// TIA Portal project "acesys_wincc_faceplates" (V16)

(* hardware
DEVICE "PC-System_1"  SIMATIC PC station
   slot 0: "SIMATIC PC station"  Rail  SIMATIC PC-Station  V1.0
      slot 125: "Stationmanager"  Station_Manager  V6.0.4
   slot 1: "HMI_RT_1"  WinCC RT Professional  6AV2 105-0xxxx-xxxx  16.0.0.0
*)

(* ===== HMI "HMI_RT_1" =====
system functions are stored by id; their names below are inferred from use
connection "994": S71200_TCP_IP, SCADA_S7_1500_OMS
connection "993": S71200_TCP_IP, SCADA_S7_1500_OMS
connection "995": S71200_TCP_IP, SCADA_S7_1500_OMS
connection "996": S71200_TCP_IP, SCADA_S7_1500_OMS
connection "997": S71200_TCP_IP, SCADA_S7_1500_OMS

HMI tags "Default tag table"
   "HMI_Tag_1" : Int, internal
   "vis_tab_int" : Int, internal
   "status_ord" : Int, internal

HMI tags "020PU043U01"
   "020PU043U01.BlockInfo" : Array [0..4] of Int AT %DB4312.DBX74.0, 500 ms
   "020PU043U01.FP_CMD" : Int AT %DB4312.DBW84, 500 ms
   "020PU043U01.FP_DIM.Auto" : Bool AT %DB4312.DBX92.0, 500 ms
   "020PU043U01.FP_DIM" : Array [0..15] of Bool AT %DB4312.DBX92.0, 500 ms
   "020PU043U01.FP_SHOW" : Array [0..15] of Bool AT %DB4312.DBX94.0, 500 ms
   "020PU043U01.FP_SHOW_1" : Int AT %DB4312.DBW96, 500 ms
   "020PU043U01.FP_SHOW.PB_Auto" : Bool AT %DB4312.DBX94.0, 500 ms
   "020PU043U01.FP_SHOW.PB_Local" : Bool AT %DB4312.DBX94.1, 500 ms
   "020PU043U01.FP_SHOW.PB_Manual" : Bool AT %DB4312.DBX94.2, 500 ms
   "020PU043U01.FP_SHOW.PB_Start1" : Bool AT %DB4312.DBX94.3, 500 ms
   "020PU043U01.FP_SHOW.PB_Start2" : Bool AT %DB4312.DBX94.4, 500 ms
   "020PU043U01.FP_SHOW.PB_Stop" : Bool AT %DB4312.DBX94.5, 500 ms
   "020PU043U01.FP_SHOW.PB_Test" : Bool AT %DB4312.DBX94.6, 500 ms
   "020PU043U01.FP_SHOW.PB_QStop" : Bool AT %DB4312.DBX94.7, 500 ms
   "020PU043U01.FP_SHOW.AI1" : Bool AT %DB4312.DBX95.0, 500 ms
   "020PU043U01.FP_SHOW.AI2" : Bool AT %DB4312.DBX95.1, 500 ms
   "020PU043U01.FP_SHOW.AI3" : Bool AT %DB4312.DBX95.2, 500 ms
   "020PU043U01.FP_SHOW.SP" : Bool AT %DB4312.DBX95.3, 500 ms
   "020PU043U01.FP_SHOW.MCC" : Bool AT %DB4312.DBX95.4, 500 ms
   "020PU043U01.FP_SHOW.RDY" : Bool AT %DB4312.DBX95.5, 500 ms
   "020PU043U01.FP_SHOW.OVL" : Bool AT %DB4312.DBX95.6, 500 ms
   "020PU043U01.FP_SHOW.LSTP" : Bool AT %DB4312.DBX95.7, 500 ms
   "020PU043U01.FP_SHOW.REM" : Bool AT %DB4312.DBX96.0, 500 ms
   "020PU043U01.FP_SHOW.SSW" : Bool AT %DB4312.DBX96.1, 500 ms
   "020PU043U01.FP_SHOW.ES" : Bool AT %DB4312.DBX96.2, 500 ms
   "020PU043U01.FP_SHOW.TFA" : Bool AT %DB4312.DBX96.3, 500 ms
   "020PU043U01.FP_SHOW.DRDY" : Bool AT %DB4312.DBX96.4, 500 ms
   "020PU043U01.FP_SHOW.STALL" : Bool AT %DB4312.DBX96.5, 500 ms
   "020PU043U01.FP_SHOW.EARTH" : Bool AT %DB4312.DBX96.6, 500 ms
   "020PU043U01.FP_SHOW.UBAL" : Bool AT %DB4312.DBX96.7, 500 ms
   "020PU043U01.FP_SHOW.GFA" : Bool AT %DB4312.DBX97.0, 500 ms
   "020PU043U01.FP_SHOW.GWA" : Bool AT %DB4312.DBX97.1, 500 ms
   "020PU043U01.FP_SHOW.BUSF" : Bool AT %DB4312.DBX97.2, 500 ms
   "020PU043U01.FP_SHOW.DOPR" : Bool AT %DB4312.DBX97.3, 500 ms
   "020PU043U01.FP_SHOW.DTEST" : Bool AT %DB4312.DBX97.4, 500 ms
   "020PU043U01.FP_SHOW.ACK" : Bool AT %DB4312.DBX97.5, 500 ms
   "020PU043U01.FP_SHOW.LSTR1" : Bool AT %DB4312.DBX97.6, 500 ms
   "020PU043U01.FP_SHOW.LSTR2" : Bool AT %DB4312.DBX97.7, 500 ms
   "020PU043U01.FP_SHOW.RET2" : Bool AT %DB4312.DBX98.0, 500 ms
   "020PU043U01.FP_SHOW.RUN2" : Bool AT %DB4312.DBX98.1, 500 ms
   "020PU043U01.FP_SHOW.CON2" : Bool AT %DB4312.DBX98.2, 500 ms
   "020PU043U01.FP_SHOW.RD2" : Bool AT %DB4312.DBX98.3, 500 ms
   "020PU043U01.FP_SHOW.SFS" : Bool AT %DB4312.DBX98.4, 500 ms
   "020PU043U01.FP_SHOW.SLS" : Bool AT %DB4312.DBX98.5, 500 ms
   "020PU043U01.FP_SHOW.MD" : Bool AT %DB4312.DBX98.6, 500 ms
   "020PU043U01.FP_SHOW.DelayRun2" : Bool AT %DB4312.DBX98.7, 500 ms
   "020PU043U01.FP_SHOW.ChangeDir" : Bool AT %DB4312.DBX99.0, 500 ms
   "020PU043U01.FP_SHOW.PB_Reset" : Bool AT %DB4312.DBX99.1, 500 ms
   "020PU043U01.FP_SHOW.ASTR" : Bool AT %DB4312.DBX99.2, 500 ms
   "020PU043U01.FP_PARM.StartWarn_Pre" : Int AT %DB4312.DBW100, 500 ms
   "020PU043U01.FP_PARM.StartWarn_Acc" : Int AT %DB4312.DBW102, 500 ms
   "020PU043U01.FP_PARM.RunDelay1_Pre" : Int AT %DB4312.DBW104, 500 ms
   "020PU043U01.FP_PARM.RunDelay1_Acc" : Int AT %DB4312.DBW106, 500 ms
   "020PU043U01.FP_PARM.RunDelay2_Pre" : Int AT %DB4312.DBW108, 500 ms
   "020PU043U01.FP_PARM.RunDelay2_Acc" : Int AT %DB4312.DBW110, 500 ms
   "020PU043U01.FP_PARM.DelayStart_Pre" : Int AT %DB4312.DBW112, 500 ms
   "020PU043U01.FP_PARM.DelayStart_Acc" : Int AT %DB4312.DBW114, 500 ms
   "020PU043U01.FP_PARM.DelayStop_Pre" : Int AT %DB4312.DBW116, 500 ms
   "020PU043U01.FP_PARM.DelayStop_Acc" : Int AT %DB4312.DBW118, 500 ms
   "020PU043U01.FP_PARM.ReturnMon_Pre" : Int AT %DB4312.DBW120, 500 ms
   "020PU043U01.FP_PARM.ReturnMon_Acc" : Int AT %DB4312.DBW122, 500 ms
   "020PU043U01.FP_PARM.SpeedMonOnDelay_Pre" : Int AT %DB4312.DBW124, 500 ms
   "020PU043U01.FP_PARM.SpeedMonOnDelay_Acc" : Int AT %DB4312.DBW126, 500 ms
   "020PU043U01.FP_PARM.SpeedMonOffDelay_Pre" : Int AT %DB4312.DBW128, 500 ms
   "020PU043U01.FP_PARM.SpeedMonOffDelay_Acc" : Int AT %DB4312.DBW130, 500 ms
   "020PU043U01.FP_PARM.SpeedMonTrigDelay_Pre" : Int AT %DB4312.DBW132, 500 ms
   "020PU043U01.FP_PARM.SpeedMonTrigDelay_Acc" : Int AT %DB4312.DBW134, 500 ms
   "020PU043U01.FP_PARM.ChangeDir_Pre" : Int AT %DB4312.DBW136, 500 ms
   "020PU043U01.FP_PARM.ChangeDir_Acc" : Int AT %DB4312.DBW138, 500 ms
   "020PU043U01.FP_PARM.LeaveFS_Pre" : Int AT %DB4312.DBW140, 500 ms
   "020PU043U01.FP_PARM.LeaveFS_Acc" : Int AT %DB4312.DBW142, 500 ms
   "020PU043U01.FP_PARM.ReachLS_Pre" : Int AT %DB4312.DBW144, 500 ms
   "020PU043U01.FP_PARM.ReachLS_Acc" : Int AT %DB4312.DBW146, 500 ms
   "020PU043U01.FP_PARM.ReachFS_Pre" : Int AT %DB4312.DBW148, 500 ms
   "020PU043U01.FP_PARM.ReachFS_Acc" : Int AT %DB4312.DBW150, 500 ms
   "020PU043U01.FP_PARM.MD_Freq_SP" : Int AT %DB4312.DBW152, 500 ms
   "020PU043U01.FP_PARM.MD_Freq_PV" : Int AT %DB4312.DBW154, 500 ms
   "020PU043U01.FP_PARM.StopReason" : Bool AT %DB4312.DBX156.0, 500 ms
   "020PU043U01.FP_PARM.AI1_Max" : Real AT %DB4312.DBD158, 500 ms
   "020PU043U01.FP_PARM.AI1_Min" : Real AT %DB4312.DBD162, 500 ms
   "020PU043U01.FP_PARM.AI2_Max" : Real AT %DB4312.DBD166, 500 ms
   "020PU043U01.FP_PARM.AI2_Min" : Real AT %DB4312.DBD170, 500 ms
   "020PU043U01.FP_PARM.AI3_Max" : Real AT %DB4312.DBD174, 500 ms
   "020PU043U01.FP_PARM.AI3_Min" : Real AT %DB4312.DBD178, 500 ms
   "020PU043U01.FP_PARM.AO1a_Max" : Real AT %DB4312.DBD182, 500 ms
   "020PU043U01.FP_PARM.AO1a_Min" : Real AT %DB4312.DBD186, 500 ms
   "020PU043U01.FP_PARM.AO2a_Max" : Real AT %DB4312.DBD190, 500 ms
   "020PU043U01.FP_PARM.AO2a_Min" : Real AT %DB4312.DBD194, 500 ms
   "020PU043U01.FP_PARM.AO3a_Max" : Real AT %DB4312.DBD198, 500 ms
   "020PU043U01.FP_PARM.AO3a_Min" : Real AT %DB4312.DBD202, 500 ms
   "020PU043U01.FP_PARM.AO1b_Max" : Real AT %DB4312.DBD206, 500 ms
   "020PU043U01.FP_PARM.AO1b_Min" : Real AT %DB4312.DBD210, 500 ms
   "020PU043U01.FP_PARM.AO2b_Max" : Real AT %DB4312.DBD214, 500 ms
   "020PU043U01.FP_PARM.AO2b_Min" : Real AT %DB4312.DBD218, 500 ms
   "020PU043U01.FP_PARM.AO3b_Max" : Real AT %DB4312.DBD222, 500 ms
   "020PU043U01.FP_PARM.AO3b_Min" : Real AT %DB4312.DBD226, 500 ms
   "020PU043U01.FP_PARM.INTL" : Bool AT %DB4312.DBX230.0, 500 ms
   "020PU043U01.FP_PARM.INTL_SEQ_STR1" : Bool AT %DB4312.DBX230.1, 500 ms
   "020PU043U01.FP_PARM.INTL_SEQ_STR2" : Bool AT %DB4312.DBX230.2, 500 ms
   "020PU043U01.FP_PARM.INTL_SEQ_STP" : Bool AT %DB4312.DBX230.3, 500 ms
   "020PU043U01.StatusWork" : Int AT %DB4312.DBW494, 500 ms
   "020PU043U01.ModePointer" : Int AT %DB4312.DBW496, 500 ms
   "020PU043U01.AO1b" : Real AT %DB4312.DBD38, 500 ms
   "020PU043U01.AO2b" : Real AT %DB4312.DBD46, 500 ms
   "020PU043U01.AO3b" : Real AT %DB4312.DBD54, 500 ms
   "020PU043U01.SPSET" : Real AT %DB4312.DBD18, 500 ms
   "020PU043U01.AO3a" : Real AT %DB4312.DBD50, 500 ms
   "020PU043U01.AO2a" : Real AT %DB4312.DBD42, 500 ms
   "020PU043U01.AO1a" : Real AT %DB4312.DBD34, 500 ms
   "020PU043U01.FP_DIM.FP_DIM" : Bool AT %DB4312.DBX92.0, 500 ms
   "020PU043U01.FP_DIM.Local" : Bool AT %DB4312.DBX92.1, 500 ms
   "020PU043U01.FP_DIM.Manual" : Bool AT %DB4312.DBX92.2, 500 ms
   "020PU043U01.FP_DIM.Start1" : Bool AT %DB4312.DBX92.3, 500 ms
   "020PU043U01.FP_DIM.Start2" : Bool AT %DB4312.DBX92.4, 500 ms
   "020PU043U01.FP_DIM.Stop" : Bool AT %DB4312.DBX92.5, 500 ms
   "020PU043U01.FP_DIM.TEst" : Bool AT %DB4312.DBX92.6, 500 ms
   "020PU043U01.FP_DIM.QStop" : Bool AT %DB4312.DBX92.7, 500 ms
   "020PU043U01.FP_DIM.Reset" : Bool AT %DB4312.DBX93.0, 500 ms
   "020PU043U01.FP_EN.Mode_Auto" : Bool AT %DB4312.DBX90.0, 500 ms
   "020PU043U01.FP_EN.Mode_Man" : Bool AT %DB4312.DBX90.1, 500 ms
   "020PU043U01.FP_EN.Mode_Loc" : Bool AT %DB4312.DBX90.2, 500 ms
   "020PU043U01.FP_EN.Mode_Test" : Bool AT %DB4312.DBX90.3, 500 ms
   "020PU043U01.FP_EN.Mode_SS_Field" : Bool AT %DB4312.DBX90.4, 500 ms
   "020PU043U01.FP_EN.Mode_SS_FP" : Bool AT %DB4312.DBX90.5, 500 ms
   "020PU043U01.FP_EN.PB_QStop" : Bool AT %DB4312.DBX90.6, 500 ms
   "020PU043U01.FP_CMD.QuickStop" : Bool AT %DB4312.DBX84.0, 500 ms
   "020PU043U01.FP_CMD.AckAlarm" : Bool AT %DB4312.DBX84.7, 500 ms
   "020PU043U01.FP_CMD.Auto" : Bool AT %DB4312.DBX85.0, 500 ms
   "020PU043U01.FP_CMD.Manual" : Bool AT %DB4312.DBX85.1, 500 ms
   "020PU043U01.FP_CMD.Local" : Bool AT %DB4312.DBX85.2, 500 ms
   "020PU043U01.FP_CMD.Start1" : Bool AT %DB4312.DBX85.3, 500 ms
   "020PU043U01.FP_CMD.Start2" : Bool AT %DB4312.DBX85.4, 500 ms
   "020PU043U01.FP_CMD.Stop" : Bool AT %DB4312.DBX85.5, 500 ms
   "020PU043U01.FP_CMD.Reset" : Bool AT %DB4312.DBX85.6, 500 ms
   "020PU043U01.FP_CMD.Test" : Bool AT %DB4312.DBX85.7, 500 ms
   "020PU043U01.DI.SEL" : Bool AT %DB4312.DBX2.0, 500 ms
   "020PU043U01.DI.ASTR" : Bool AT %DB4312.DBX2.1, 500 ms
   "020PU043U01.DI.DIR" : Bool AT %DB4312.DBX2.2, 500 ms
   "020PU043U01.DI.MCC" : Bool AT %DB4312.DBX2.3, 500 ms
   "020PU043U01.DI.RDY" : Bool AT %DB4312.DBX2.4, 500 ms
   "020PU043U01.DI.OVL" : Bool AT %DB4312.DBX2.5, 500 ms
   "020PU043U01.DI.RET1" : Bool AT %DB4312.DBX2.6, 500 ms
   "020PU043U01.DI.RET2" : Bool AT %DB4312.DBX2.7, 500 ms
   "020PU043U01.DI.LSTR1" : Bool AT %DB4312.DBX3.0, 500 ms
   "020PU043U01.DI.LSTR2" : Bool AT %DB4312.DBX3.1, 500 ms
   "020PU043U01.DI.LSTP" : Bool AT %DB4312.DBX3.2, 500 ms
   "020PU043U01.DI.REM" : Bool AT %DB4312.DBX3.3, 500 ms
   "020PU043U01.DI.SSW" : Bool AT %DB4312.DBX3.4, 500 ms
   "020PU043U01.DI.TFA" : Bool AT %DB4312.DBX3.5, 500 ms
   "020PU043U01.DI.DRDY" : Bool AT %DB4312.DBX3.6, 500 ms
   "020PU043U01.DI.MD" : Bool AT %DB4312.DBX3.7, 500 ms
   "020PU043U01.DI.STALL" : Bool AT %DB4312.DBX4.0, 500 ms
   "020PU043U01.DI.EARTH" : Bool AT %DB4312.DBX4.1, 500 ms
   "020PU043U01.DI.UBAL" : Bool AT %DB4312.DBX4.2, 500 ms
   "020PU043U01.DI.GFA" : Bool AT %DB4312.DBX4.3, 500 ms
   "020PU043U01.DI.GWA" : Bool AT %DB4312.DBX4.4, 500 ms
   "020PU043U01.DI.BUSF" : Bool AT %DB4312.DBX4.5, 500 ms
   "020PU043U01.DI.DOPR" : Bool AT %DB4312.DBX4.6, 500 ms
   "020PU043U01.DI.DTEST" : Bool AT %DB4312.DBX4.7, 500 ms
   "020PU043U01.DI.SFS" : Bool AT %DB4312.DBX5.0, 500 ms
   "020PU043U01.DI.SLS" : Bool AT %DB4312.DBX5.1, 500 ms
   "020PU043U01.DI.ES" : Bool AT %DB4312.DBX5.2, 500 ms
   "020PU043U01.DI.ACK" : Bool AT %DB4312.DBX5.3, 500 ms
   "020PU043U01.DQ.CON1" : Bool AT %DB4312.DBX30.0, 500 ms
   "020PU043U01.DQ.CON2" : Bool AT %DB4312.DBX30.1, 500 ms
   "020PU043U01.DQ.LAMP1" : Bool AT %DB4312.DBX30.2, 500 ms
   "020PU043U01.DQ.LAMP2" : Bool AT %DB4312.DBX30.3, 500 ms
   "020PU043U01.DQ.SACK" : Bool AT %DB4312.DBX30.4, 500 ms
   "020PU043U01.DQ.RD1" : Bool AT %DB4312.DBX30.5, 500 ms
   "020PU043U01.DQ.RD2" : Bool AT %DB4312.DBX30.6, 500 ms
   "020PU043U01.DQ.RUN1" : Bool AT %DB4312.DBX30.7, 500 ms
   "020PU043U01.DQ.RUN2" : Bool AT %DB4312.DBX31.0, 500 ms
   "020PU043U01.DQ.OK" : Bool AT %DB4312.DBX31.1, 500 ms
   "020PU043U01.DQ.LOC" : Bool AT %DB4312.DBX31.2, 500 ms
   "020PU043U01.DQ.MAN" : Bool AT %DB4312.DBX31.3, 500 ms
   "020PU043U01.DQ.AUT" : Bool AT %DB4312.DBX31.4, 500 ms
   "020PU043U01.DQ.SS" : Bool AT %DB4312.DBX31.5, 500 ms
   "020PU043U01.DQ.RES" : Bool AT %DB4312.DBX31.6, 500 ms
   "020PU043U01.DQ.TESTP" : Bool AT %DB4312.DBX31.7, 500 ms
   "020PU043U01.DQ.ASTW" : Bool AT %DB4312.DBX32.0, 500 ms
   "020PU043U01.AI1" : Real AT %DB4312.DBD6, 500 ms
   "020PU043U01.AI2" : Real AT %DB4312.DBD10, 500 ms
   "020PU043U01.AI3" : Real AT %DB4312.DBD14, 500 ms
   "020PU043U01.FP_SEL.MD" : Bool AT %DB4312.DBX86.0, 500 ms
   "020PU043U01.FP_SEL.MD_Puls" : Bool AT %DB4312.DBX86.1, 500 ms
   "020PU043U01.FP_SEL.MD_OnOff" : Bool AT %DB4312.DBX86.2, 500 ms
   "020PU043U01.FP_SEL.MD_Maintain" : Bool AT %DB4312.DBX86.3, 500 ms
   "020PU043U01.FP_SEL.STW_AutoStart" : Bool AT %DB4312.DBX86.4, 500 ms
   "020PU043U01.FP_SEL.STW_Local" : Bool AT %DB4312.DBX86.5, 500 ms
   "020PU043U01.FP_SEL.STW_Manual" : Bool AT %DB4312.DBX86.6, 500 ms
   "020PU043U01.FP_SEL.STW_Single" : Bool AT %DB4312.DBX86.7, 500 ms
   "020PU043U01.FP_SEL.Type_Unimotor" : Bool AT %DB4312.DBX87.0, 500 ms
   "020PU043U01.FP_SEL.Type_Bimotor" : Bool AT %DB4312.DBX87.1, 500 ms
   "020PU043U01.FP_SEL.Type_Indication" : Bool AT %DB4312.DBX87.2, 500 ms
   "020PU043U01.FP_SEL.MotorStarter" : Bool AT %DB4312.DBX87.3, 500 ms
   "020PU043U01.FP_SEL.ParentSupress" : Bool AT %DB4312.DBX87.4, 500 ms
   "020PU043U01.FP_SEL.ParentCollection" : Bool AT %DB4312.DBX87.5, 500 ms
   "020PU043U01.FP_SEL.INCH_Man" : Bool AT %DB4312.DBX87.6, 500 ms
   "020PU043U01.FP_SEL.INCH_Loc" : Bool AT %DB4312.DBX87.7, 500 ms
   "020PU043U01.FP_SEL.OutOfSevice" : Bool AT %DB4312.DBX88.0, 500 ms
   "020PU043U01.FP_SEL.WarningDrive" : Bool AT %DB4312.DBX88.1, 500 ms
   "020PU043U01.FP_SHOW.B1" : Byte AT %DB4313.DBB95, 500 ms
   "020PU043U01.FP_SHOW.B2" : Byte AT %DB4313.DBB96, 500 ms
   "020PU043U01.FP_SHOW.B3" : Byte AT %DB4313.DBB97, 500 ms
   "020PU043U01.FP_SHOW.B4" : Byte AT %DB4313.DBB98, 500 ms
   "020PU043U01.FP_SHOW.B5" : Byte AT %DB4313.DBB99, 500 ms
   "020PU043U01.MSW" : DWord AT %DB4312.DBD62, 500 ms
   "020PU043U01.ParentInfo" : String[10], internal
   "020PU043U01.DefaultText" : String[32], internal   // Заголовок POPUP окна. При експорте из ECS через скрипт заполняется автоматически, если теги копируются в ручную то требуется в ручную задатать свойство Start Value

HMI tags "020PU044U01"
   "020PU044U01.BlockInfo" : Array [0..4] of Int AT %DB4313.DBX74.0, 500 ms
   "020PU044U01.FP_CMD" : Int AT %DB4313.DBW84, 500 ms
   "020PU044U01.MSW" : DWord AT %DB4313.DBD62, 500 ms
   "020PU044U01.FP_DIM.Auto" : Bool AT %DB4313.DBX92.0, 500 ms
   "020PU044U01.FP_DIM1" : Array [0..15] of Bool AT %DB4313.DBX92.0, 500 ms
   "020PU044U01.FP_SHOW" : Array [0..15] of Bool AT %DB4313.DBX94.0, 500 ms
   "020PU044U01.FP_SHOW_1" : Int AT %DB4313.DBW96, 500 ms
   "020PU044U01.FP_SHOW.PB_Auto" : Bool AT %DB4313.DBX94.0, 500 ms
   "020PU044U01.FP_SHOW.PB_Local" : Bool AT %DB4313.DBX94.1, 500 ms
   "020PU044U01.FP_SHOW.PB_Manual" : Bool AT %DB4313.DBX94.2, 500 ms
   "020PU044U01.FP_SHOW.PB_Start1" : Bool AT %DB4313.DBX94.3, 500 ms
   "020PU044U01.FP_SHOW.PB_Start2" : Bool AT %DB4313.DBX94.4, 500 ms
   "020PU044U01.FP_SHOW.PB_Stop" : Bool AT %DB4313.DBX94.5, 500 ms
   "020PU044U01.FP_SHOW.PB_Test" : Bool AT %DB4313.DBX94.6, 500 ms
   "020PU044U01.FP_SHOW.PB_QStop" : Bool AT %DB4313.DBX94.7, 500 ms
   "020PU044U01.FP_SHOW.AI1" : Bool AT %DB4313.DBX95.0, 500 ms
   "020PU044U01.FP_SHOW.AI2" : Bool AT %DB4313.DBX95.1, 500 ms
   "020PU044U01.FP_SHOW.AI3" : Bool AT %DB4313.DBX95.2, 500 ms
   "020PU044U01.FP_SHOW.SP" : Bool AT %DB4313.DBX95.3, 500 ms
   "020PU044U01.FP_SHOW.MCC" : Bool AT %DB4313.DBX95.4, 500 ms
   "020PU044U01.FP_SHOW.RDY" : Bool AT %DB4313.DBX95.5, 500 ms
   "020PU044U01.FP_SHOW.OVL" : Bool AT %DB4313.DBX95.6, 500 ms
   "020PU044U01.FP_SHOW.LSTP" : Bool AT %DB4313.DBX95.7, 500 ms
   "020PU044U01.FP_SHOW.REM" : Bool AT %DB4313.DBX96.0, 500 ms
   "020PU044U01.FP_SHOW.SSW" : Bool AT %DB4313.DBX96.1, 500 ms
   "020PU044U01.FP_SHOW.ES" : Bool AT %DB4313.DBX96.2, 500 ms
   "020PU044U01.FP_SHOW.TFA" : Bool AT %DB4313.DBX96.3, 500 ms
   "020PU044U01.FP_SHOW.DRDY" : Bool AT %DB4313.DBX96.4, 500 ms
   "020PU044U01.FP_SHOW.STALL" : Bool AT %DB4313.DBX96.5, 500 ms
   "020PU044U01.FP_SHOW.EARTH" : Bool AT %DB4313.DBX96.6, 500 ms
   "020PU044U01.FP_SHOW.UBAL" : Bool AT %DB4313.DBX96.7, 500 ms
   "020PU044U01.FP_SHOW.GFA" : Bool AT %DB4313.DBX97.0, 500 ms
   "020PU044U01.FP_SHOW.GWA" : Bool AT %DB4313.DBX97.1, 500 ms
   "020PU044U01.FP_SHOW.BUSF" : Bool AT %DB4313.DBX97.2, 500 ms
   "020PU044U01.FP_SHOW.DOPR" : Bool AT %DB4313.DBX97.3, 500 ms
   "020PU044U01.FP_SHOW.DTEST" : Bool AT %DB4313.DBX97.4, 500 ms
   "020PU044U01.FP_SHOW.ACK" : Bool AT %DB4313.DBX97.5, 500 ms
   "020PU044U01.FP_SHOW.LSTR1" : Bool AT %DB4313.DBX97.6, 500 ms
   "020PU044U01.FP_SHOW.LSTR2" : Bool AT %DB4313.DBX97.7, 500 ms
   "020PU044U01.FP_SHOW.RET2" : Bool AT %DB4313.DBX98.0, 500 ms
   "020PU044U01.FP_SHOW.RUN2" : Bool AT %DB4313.DBX98.1, 500 ms
   "020PU044U01.FP_SHOW.CON2" : Bool AT %DB4313.DBX98.2, 500 ms
   "020PU044U01.FP_SHOW.RD2" : Bool AT %DB4313.DBX98.3, 500 ms
   "020PU044U01.FP_SHOW.SFS" : Bool AT %DB4313.DBX98.4, 500 ms
   "020PU044U01.FP_SHOW.SLS" : Bool AT %DB4313.DBX98.5, 500 ms
   "020PU044U01.FP_SHOW.MD" : Bool AT %DB4313.DBX98.6, 500 ms
   "020PU044U01.FP_SHOW.DelayRun2" : Bool AT %DB4313.DBX98.7, 500 ms
   "020PU044U01.FP_SHOW.ChangeDir" : Bool AT %DB4313.DBX99.0, 500 ms
   "020PU044U01.FP_SHOW.PB_Reset" : Bool AT %DB4313.DBX99.1, 500 ms
   "020PU044U01.FP_SHOW.ASTR" : Bool AT %DB4313.DBX99.2, 500 ms
   "020PU044U01.FP_PARM.StartWarn_Pre" : Int AT %DB4313.DBW100, 500 ms
   "020PU044U01.FP_PARM.StartWarn_Acc" : Int AT %DB4313.DBW102, 500 ms
   "020PU044U01.FP_PARM.RunDelay1_Pre" : Int AT %DB4313.DBW104, 500 ms
   "020PU044U01.FP_PARM.RunDelay1_Acc" : Int AT %DB4313.DBW106, 500 ms
   "020PU044U01.FP_PARM.RunDelay2_Pre" : Int AT %DB4313.DBW108, 500 ms
   "020PU044U01.FP_PARM.RunDelay2_Acc" : Int AT %DB4313.DBW110, 500 ms
   "020PU044U01.FP_PARM.DelayStart_Pre" : Int AT %DB4313.DBW112, 500 ms
   "020PU044U01.FP_PARM.DelayStart_Acc" : Int AT %DB4313.DBW114, 500 ms
   "020PU044U01.FP_PARM.DelayStop_Pre" : Int AT %DB4313.DBW116, 500 ms
   "020PU044U01.FP_PARM.DelayStop_Acc" : Int AT %DB4313.DBW118, 500 ms
   "020PU044U01.FP_PARM.ReturnMon_Pre" : Int AT %DB4313.DBW120, 500 ms
   "020PU044U01.FP_PARM.ReturnMon_Acc" : Int AT %DB4313.DBW122, 500 ms
   "020PU044U01.FP_PARM.SpeedMonOnDelay_Pre" : Int AT %DB4313.DBW124, 500 ms
   "020PU044U01.FP_PARM.SpeedMonOnDelay_Acc" : Int AT %DB4313.DBW126, 500 ms
   "020PU044U01.FP_PARM.SpeedMonOffDelay_Pre" : Int AT %DB4313.DBW128, 500 ms
   "020PU044U01.FP_PARM.SpeedMonOffDelay_Acc" : Int AT %DB4313.DBW130, 500 ms
   "020PU044U01.FP_PARM.SpeedMonTrigDelay_Pre" : Int AT %DB4313.DBW132, 500 ms
   "020PU044U01.FP_PARM.SpeedMonTrigDelay_Acc" : Int AT %DB4313.DBW134, 500 ms
   "020PU044U01.FP_PARM.ChangeDir_Pre" : Int AT %DB4313.DBW136, 500 ms
   "020PU044U01.FP_PARM.ChangeDir_Acc" : Int AT %DB4313.DBW138, 500 ms
   "020PU044U01.FP_PARM.LeaveFS_Pre" : Int AT %DB4313.DBW140, 500 ms
   "020PU044U01.FP_PARM.LeaveFS_Acc" : Int AT %DB4313.DBW142, 500 ms
   "020PU044U01.FP_PARM.ReachLS_Pre" : Int AT %DB4313.DBW144, 500 ms
   "020PU044U01.FP_PARM.ReachLS_Acc" : Int AT %DB4313.DBW146, 500 ms
   "020PU044U01.FP_PARM.ReachFS_Pre" : Int AT %DB4313.DBW148, 500 ms
   "020PU044U01.FP_PARM.ReachFS_Acc" : Int AT %DB4313.DBW150, 500 ms
   "020PU044U01.FP_PARM.MD_Freq_SP" : Int AT %DB4313.DBW152, 500 ms
   "020PU044U01.FP_PARM.MD_Freq_PV" : Int AT %DB4313.DBW154, 500 ms
   "020PU044U01.FP_PARM.StopReason" : Int AT %DB4313.DBW156, 500 ms
   "020PU044U01.FP_PARM.AI1_Max" : Real AT %DB4313.DBD158, 500 ms
   "020PU044U01.FP_PARM.AI1_Min" : Real AT %DB4313.DBD162, 500 ms
   "020PU044U01.FP_PARM.AI2_Max" : Real AT %DB4313.DBD166, 500 ms
   "020PU044U01.FP_PARM.AI2_Min" : Real AT %DB4313.DBD170, 500 ms
   "020PU044U01.FP_PARM.AI3_Max" : Real AT %DB4313.DBD174, 500 ms
   "020PU044U01.FP_PARM.AI3_Min" : Real AT %DB4313.DBD178, 500 ms
   "020PU044U01.FP_PARM.AO1a_Max" : Real AT %DB4313.DBD182, 500 ms
   "020PU044U01.FP_PARM.AO1a_Min" : Real AT %DB4313.DBD186, 500 ms
   "020PU044U01.FP_PARM.AO2a_Max" : Real AT %DB4313.DBD190, 500 ms
   "020PU044U01.FP_PARM.AO2a_Min" : Real AT %DB4313.DBD194, 500 ms
   "020PU044U01.FP_PARM.AO3a_Max" : Real AT %DB4313.DBD198, 500 ms
   "020PU044U01.FP_PARM.AO3a_Min" : Real AT %DB4313.DBD202, 500 ms
   "020PU044U01.FP_PARM.AO1b_Max" : Real AT %DB4313.DBD206, 500 ms
   "020PU044U01.FP_PARM.AO1b_Min" : Real AT %DB4313.DBD210, 500 ms
   "020PU044U01.FP_PARM.AO2b_Max" : Real AT %DB4313.DBD214, 500 ms
   "020PU044U01.FP_PARM.AO2b_Min" : Real AT %DB4313.DBD218, 500 ms
   "020PU044U01.FP_PARM.AO3b_Max" : Real AT %DB4313.DBD222, 500 ms
   "020PU044U01.FP_PARM.AO3b_Min" : Real AT %DB4313.DBD226, 500 ms
   "020PU044U01.FP_PARM.INTL" : Bool AT %DB4313.DBX230.0, 500 ms
   "020PU044U01.FP_PARM.INTL_SEQ_STR1" : Bool AT %DB4313.DBX230.1, 500 ms
   "020PU044U01.FP_PARM.INTL_SEQ_STR2" : Bool AT %DB4313.DBX230.2, 500 ms
   "020PU044U01.FP_PARM.INTL_SEQ_STP" : Bool AT %DB4313.DBX230.3, 500 ms
   "020PU044U01.StatusWork" : Int AT %DB4313.DBW494, 500 ms
   "020PU044U01.ModePointer" : Int AT %DB4313.DBW496, 500 ms
   "020PU044U01.AO1b" : Real AT %DB4313.DBD38, 500 ms
   "020PU044U01.AO2b" : Real AT %DB4313.DBD42, 500 ms
   "020PU044U01.AO3b" : Real AT %DB4313.DBD46, 500 ms
   "020PU044U01.SPSET" : Real AT %DB4313.DBD18, 500 ms
   "020PU044U01.AO3a" : Real AT %DB4313.DBD50, 500 ms
   "020PU044U01.AO2a" : Real AT %DB4313.DBD42, 500 ms
   "020PU044U01.AO1a" : Real AT %DB4313.DBD34, 500 ms
   "020PU044U01.FP_DIM.FP_DIM" : Bool AT %DB4313.DBX92.0, 500 ms
   "020PU044U01.FP_DIM.Local" : Bool AT %DB4313.DBX92.1, 500 ms
   "020PU044U01.FP_DIM.Manual" : Bool AT %DB4313.DBX92.2, 500 ms
   "020PU044U01.FP_DIM.Start1" : Bool AT %DB4313.DBX92.3, 500 ms
   "020PU044U01.FP_DIM.Start2" : Bool AT %DB4313.DBX92.4, 500 ms
   "020PU044U01.FP_DIM.Stop" : Bool AT %DB4313.DBX92.5, 500 ms
   "020PU044U01.FP_DIM.TEst" : Bool AT %DB4313.DBX92.6, 500 ms
   "020PU044U01.FP_DIM.QStop" : Bool AT %DB4313.DBX92.7, 500 ms
   "020PU044U01.FP_DIM.Reset" : Bool AT %DB4313.DBX93.0, 500 ms
   "020PU044U01.FP_EN.Mode_Auto" : Bool AT %DB4313.DBX90.0, 500 ms
   "020PU044U01.FP_EN.Mode_Man" : Bool AT %DB4313.DBX90.1, 500 ms
   "020PU044U01.FP_EN.Mode_Loc" : Bool AT %DB4313.DBX90.2, 500 ms
   "020PU044U01.FP_EN.Mode_Test" : Bool AT %DB4313.DBX90.3, 500 ms
   "020PU044U01.FP_EN.Mode_SS_Field" : Bool AT %DB4313.DBX90.4, 500 ms
   "020PU044U01.FP_EN.Mode_SS_FP" : Bool AT %DB4313.DBX90.5, 500 ms
   "020PU044U01.FP_EN.PB_QStop" : Bool AT %DB4313.DBX90.6, 500 ms
   "020PU044U01.FP_EN.Mode_Loc_1" : Bool AT %DB4313.DBX90.3, 500 ms
   "020PU044U01.FP_CMD.QuickStop" : Bool AT %DB4313.DBX84.0, 500 ms
   "020PU044U01.FP_CMD.AckAlarm" : Bool AT %DB4313.DBX84.7, 500 ms
   "020PU044U01.FP_CMD.Auto" : Bool AT %DB4313.DBX85.0, 500 ms
   "020PU044U01.FP_CMD.Manual" : Bool AT %DB4313.DBX85.1, 500 ms
   "020PU044U01.FP_CMD.Local" : Bool AT %DB4313.DBX85.2, 500 ms
   "020PU044U01.FP_CMD.Start1" : Bool AT %DB4313.DBX85.3, 500 ms
   "020PU044U01.FP_CMD.Start2" : Bool AT %DB4313.DBX85.4, 500 ms
   "020PU044U01.FP_CMD.Stop" : Bool AT %DB4313.DBX85.5, 500 ms
   "020PU044U01.FP_CMD.Reset" : Bool AT %DB4313.DBX85.6, 500 ms
   "020PU044U01.FP_CMD.Test" : Bool AT %DB4313.DBX85.7, 500 ms
   "020PU044U01.DI.SEL" : Bool AT %DB4313.DBX2.0, 500 ms
   "020PU044U01.DI.ASTR" : Bool AT %DB4313.DBX2.1, 500 ms
   "020PU044U01.DI.DIR" : Bool AT %DB4313.DBX2.2, 500 ms
   "020PU044U01.DI.MCC" : Bool AT %DB4313.DBX2.3, 500 ms
   "020PU044U01.DI.RDY" : Bool AT %DB4313.DBX2.4, 500 ms
   "020PU044U01.DI.OVL" : Bool AT %DB4313.DBX2.5, 500 ms
   "020PU044U01.DI.RET1" : Bool AT %DB4313.DBX2.6, 500 ms
   "020PU044U01.DI.RET2" : Bool AT %DB4313.DBX2.7, 500 ms
   "020PU044U01.DI.LSTR1" : Bool AT %DB4313.DBX3.0, 500 ms
   "020PU044U01.DI.LSTR2" : Bool AT %DB4313.DBX3.1, 500 ms
   "020PU044U01.DI.LSTP" : Bool AT %DB4313.DBX3.2, 500 ms
   "020PU044U01.DI.REM" : Bool AT %DB4313.DBX3.3, 500 ms
   "020PU044U01.DI.SSW" : Bool AT %DB4313.DBX3.4, 500 ms
   "020PU044U01.DI.TFA" : Bool AT %DB4313.DBX3.5, 500 ms
   "020PU044U01.DI.DRDY" : Bool AT %DB4313.DBX3.6, 500 ms
   "020PU044U01.DI.MD" : Bool AT %DB4313.DBX3.7, 500 ms
   "020PU044U01.DI.STALL" : Bool AT %DB4313.DBX4.0, 500 ms
   "020PU044U01.DI.EARTH" : Bool AT %DB4313.DBX4.1, 500 ms
   "020PU044U01.DI.UBAL" : Bool AT %DB4313.DBX4.2, 500 ms
   "020PU044U01.DI.GFA" : Bool AT %DB4313.DBX4.3, 500 ms
   "020PU044U01.DI.GWA" : Bool AT %DB4313.DBX4.4, 500 ms
   "020PU044U01.DI.BUSF" : Bool AT %DB4313.DBX4.5, 500 ms
   "020PU044U01.DI.DOPR" : Bool AT %DB4313.DBX4.6, 500 ms
   "020PU044U01.DI.DTEST" : Bool AT %DB4313.DBX4.7, 500 ms
   "020PU044U01.DI.SFS" : Bool AT %DB4313.DBX5.0, 500 ms
   "020PU044U01.DI.SLS" : Bool AT %DB4313.DBX5.1, 500 ms
   "020PU044U01.DI.ES" : Bool AT %DB4313.DBX5.2, 500 ms
   "020PU044U01.DI.ACK" : Bool AT %DB4313.DBX5.3, 500 ms
   "020PU044U01.DQ.CON1" : Bool AT %DB4313.DBX30.0, 500 ms
   "020PU044U01.DQ.CON2" : Bool AT %DB4313.DBX30.1, 500 ms
   "020PU044U01.DQ.LAMP1" : Bool AT %DB4313.DBX30.2, 500 ms
   "020PU044U01.DQ.LAMP2" : Bool AT %DB4313.DBX30.3, 500 ms
   "020PU044U01.DQ.SACK" : Bool AT %DB4313.DBX30.4, 500 ms
   "020PU044U01.DQ.RD1" : Bool AT %DB4313.DBX30.5, 500 ms
   "020PU044U01.DQ.RD2" : Bool AT %DB4313.DBX30.6, 500 ms
   "020PU044U01.DQ.RUN1" : Bool AT %DB4313.DBX30.7, 500 ms
   "020PU044U01.DQ.RUN2" : Bool AT %DB4313.DBX31.0, 500 ms
   "020PU044U01.DQ.OK" : Bool AT %DB4313.DBX31.1, 500 ms
   "020PU044U01.DQ.LOC" : Bool AT %DB4313.DBX31.2, 500 ms
   "020PU044U01.DQ.MAN" : Bool AT %DB4313.DBX31.3, 500 ms
   "020PU044U01.DQ.AUT" : Bool AT %DB4313.DBX31.4, 500 ms
   "020PU044U01.DQ.SS" : Bool AT %DB4313.DBX31.5, 500 ms
   "020PU044U01.DQ.RES" : Bool AT %DB4313.DBX31.6, 500 ms
   "020PU044U01.DQ.TESTP" : Bool AT %DB4313.DBX31.7, 500 ms
   "020PU044U01.DQ.ASTW" : Bool AT %DB4313.DBX32.0, 500 ms
   "020PU044U01.AI1" : Real AT %DB4313.DBD6, 500 ms
   "020PU044U01.AI2" : Real AT %DB4313.DBD10, 500 ms
   "020PU044U01.AI3" : Real AT %DB4313.DBD14, 500 ms
   "020PU044U01.FP_SEL.MD" : Bool AT %DB4313.DBX86.0, 500 ms
   "020PU044U01.FP_SEL.MD_Puls" : Bool AT %DB4313.DBX86.1, 500 ms
   "020PU044U01.FP_SEL.MD_OnOff" : Bool AT %DB4313.DBX86.2, 500 ms
   "020PU044U01.FP_SEL.MD_Maintain" : Bool AT %DB4313.DBX86.3, 500 ms
   "020PU044U01.FP_SEL.STW_AutoStart" : Bool AT %DB4313.DBX86.4, 500 ms
   "020PU044U01.FP_SEL.STW_Local" : Bool AT %DB4313.DBX86.5, 500 ms
   "020PU044U01.FP_SEL.STW_Manual" : Bool AT %DB4313.DBX86.6, 500 ms
   "020PU044U01.FP_SEL.STW_Single" : Bool AT %DB4313.DBX86.7, 500 ms
   "020PU044U01.FP_SEL.Type_Unimotor" : Bool AT %DB4313.DBX87.0, 500 ms
   "020PU044U01.FP_SEL.Type_Bimotor" : Bool AT %DB4313.DBX87.1, 500 ms
   "020PU044U01.FP_SEL.Type_Indication" : Bool AT %DB4313.DBX87.2, 500 ms
   "020PU044U01.FP_SEL.MotorStarter" : Bool AT %DB4313.DBX87.3, 500 ms
   "020PU044U01.FP_SEL.ParentSupress" : Bool AT %DB4313.DBX87.4, 500 ms
   "020PU044U01.FP_SEL.ParentCollection" : Bool AT %DB4313.DBX87.5, 500 ms
   "020PU044U01.FP_SEL.INCH_Man" : Bool AT %DB4313.DBX87.6, 500 ms
   "020PU044U01.FP_SEL.INCH_Loc" : Bool AT %DB4313.DBX87.7, 500 ms
   "020PU044U01.FP_SEL.OutOfSevice" : Bool AT %DB4313.DBX88.0, 500 ms
   "020PU044U01.FP_SEL.WarningDrive" : Bool AT %DB4313.DBX88.1, 500 ms
   "020PU044U01.FP_SHOW.B1" : Byte AT %DB4313.DBB95, 500 ms
   "020PU044U01.FP_SHOW.B2" : Byte AT %DB4313.DBB96, 500 ms
   "020PU044U01.FP_SHOW.B3" : Byte AT %DB4313.DBB97, 500 ms
   "020PU044U01.FP_SHOW.B4" : Byte AT %DB4313.DBB98, 500 ms
   "msw_stuct" : aaebc164-1e5c-4a03-9189-7c4808a568f8 AT %DB4313.DBX62.0, 500 ms
   "020PU044U01.ParentInfo" : TextRef, internal   // Имя родителя для попап окна, вкладка инфо. При експорте из ECS через скрипт заполняется автоматически, если теги копируются в ручную то требуется в ручную задатать свойство Start Value
   "020PU044U01.DefaultText" : TextRef, internal   // Заголовок POPUP окна. При експорте из ECS через скрипт заполняется автоматически, если теги копируются в ручную то требуется в ручную задатать свойство Start Value
   "020PU044U01.INTL01" : Byte AT %DB10.DBB316, 500 ms   // Interlock
   "020PU044U01.INTL01.DefaultText" : TextRef, internal
   "020PU044U01.STR01" : Byte AT %DB10.DBB317, 500 ms
   "020PU044U01.STR01.DefaultText" : TextRef, internal   // Sequence Interlocking
   "020PU044U01.STP01" : Byte AT %DB10.DBB320, 500 ms   // Sequence Stop Enable
   "020PU044U01.STP01.DefaultText" : TextRef, internal   // Sequence Stop Enable

HMI tags "utils"
   "cursor_pos_x" : Int, internal
   "cursor_pos_y" : Int, internal
   "temp_int" : Int, internal
   "tmp_bool" : Bool, internal

HMI tags "Internal_Tag"
   "Control_FP" : Int, internal
   "Realyted_Point_FP" : Int, internal
   "Input_FP" : Int, internal
   "Output_FP" : Int, internal
   "Timers_FP" : Int, internal

HMI tags "2080SP241U01S01"
   "2080SP241U01S01.MSW" : 52809b66-421d-457f-8884-6f7a49d4e247 AT %DB5289.DBX18.0, 500 ms
   "2080SP241U01S01.ParentInfo" : TextRef, internal   // Имя родителя для попап окна, вкладка инфо. При експорте из ECS через скрипт заполняется автоматически, если теги копируются в ручную то требуется в ручную задатать свойство Start Value
   "2080SP241U01S01.DefaultText" : TextRef, internal   // Заголовок POPUP окна. При експорте из ECS через скрипт заполняется автоматически, если теги копируются в ручную то требуется в ручную задатать свойство Start Value
   "2080SP241U01S01.BlockInfo" : Array [0..2] of Int AT %DB5289.DBX38.0, 500 ms
   "2080SP241U01S01.StatusWork" : Int AT %DB5289.DBW242, 500 ms
   "2080SP241U01S01.FP_PARAM.DampingTime" : Int AT %DB5289.DBW50, 500 ms
   "2080SP241U01S01.FP_PARAM.Force_Value" : Real AT %DB5289.DBD52, 500 ms
   "2080SP241U01S01.FP_PARAM.Scale_Min" : Real AT %DB5289.DBD56, 500 ms
   "2080SP241U01S01.FP_PARAM.Scale_Max" : Real AT %DB5289.DBD60, 500 ms
   "2080SP241U01S01.FP_PARAM.Gradient" : Real AT %DB5289.DBD64, 500 ms
   "2080SP241U01S01.FP_PARAM.Grad_Pos" : Real AT %DB5289.DBD68, 500 ms
   "2080SP241U01S01.FP_PARAM.Grad_Neg" : Real AT %DB5289.DBD72, 500 ms
   "2080SP241U01S01.FP_PARAM.Grad_X" : Real AT %DB5289.DBD76, 500 ms
   "2080SP241U01S01.FP_PARAM.Gradient_Time_Pre" : Int AT %DB5289.DBW80, 500 ms
   "2080SP241U01S01.FP_PARAM.Gradient_Time_ACC" : Int AT %DB5289.DBW82, 500 ms
   "2080SP241U01S01.FP_PARAM.Alarm_Hyst" : Real AT %DB5289.DBD84, 500 ms
   "2080SP241U01S01.FP_PARAM.AlarmLimit_H3" : Real AT %DB5289.DBD88, 500 ms
   "2080SP241U01S01.FP_PARAM.AlarmLimit_H2" : Real AT %DB5289.DBD92, 500 ms
   "2080SP241U01S01.FP_PARAM.AlarmLimit_H1" : Real AT %DB5289.DBD96, 500 ms
   "2080SP241U01S01.FP_PARAM.AlarmLimit_L1" : Real AT %DB5289.DBD100, 500 ms
   "2080SP241U01S01.FP_PARAM.AlarmLimit_L2" : Real AT %DB5289.DBD104, 500 ms
   "2080SP241U01S01.FP_PARAM.AlarmLimit_L3" : Real AT %DB5289.DBD108, 500 ms
   "2080SP241U01S01.FP_PARAM.AlarmDelay_H3_Pre" : Int AT %DB5289.DBW112, 500 ms
   "2080SP241U01S01.FP_PARAM.AlarmDelay_H3_Acc" : Int AT %DB5289.DBW114, 500 ms
   "2080SP241U01S01.FP_PARAM.AlarmDelay_H2_Pre" : Int AT %DB5289.DBW116, 500 ms
   "2080SP241U01S01.FP_PARAM.AlarmDelay_H2_Acc" : Int AT %DB5289.DBW118, 500 ms
   "2080SP241U01S01.FP_PARAM.AlarmDelay_H1_Pre" : Int AT %DB5289.DBW120, 500 ms
   "2080SP241U01S01.FP_PARAM.AlarmDelay_H1_Acc" : Int AT %DB5289.DBW122, 500 ms
   "2080SP241U01S01.FP_PARAM.AlarmDelay_L1_Pre" : Int AT %DB5289.DBW124, 500 ms
   "2080SP241U01S01.FP_PARAM.AlarmDelay_L1_Acc" : Int AT %DB5289.DBW126, 500 ms
   "2080SP241U01S01.FP_PARAM.AlarmDelay_L2_Pre" : Int AT %DB5289.DBW128, 500 ms
   "2080SP241U01S01.FP_PARAM.AlarmDelay_L2_Acc" : Int AT %DB5289.DBW130, 500 ms
   "2080SP241U01S01.FP_PARAM.AlarmDelay_L3_Pre" : Int AT %DB5289.DBW132, 500 ms
   "2080SP241U01S01.FP_PARAM.AlarmDelay_L3_Acc" : Int AT %DB5289.DBW134, 500 ms
   "2080SP241U01S01.FP_PARAM.OpenLoopDelay_Pre" : Int AT %DB5289.DBW136, 500 ms
   "2080SP241U01S01.FP_PARAM.OpenLoopDelay_Acc" : Int AT %DB5289.DBW138, 500 ms
   "2080SP241U01S01.FP_PARAM.OverRangeDelay_Pre" : Int AT %DB5289.DBW140, 500 ms
   "2080SP241U01S01.FP_PARAM.OverRangeDelay_Acc" : Int AT %DB5289.DBW142, 500 ms
   "2080SP241U01S01.FP_PARAM.AuxLimit_H2_Value" : Real AT %DB5289.DBD144, 500 ms
   "2080SP241U01S01.FP_PARAM.AuxLimit_H1_Value" : Real AT %DB5289.DBD148, 500 ms
   "2080SP241U01S01.FP_PARAM.AuxLimit_L2_Value" : Real AT %DB5289.DBD152, 500 ms
   "2080SP241U01S01.FP_PARAM.AuxLimit_L1_Value" : Real AT %DB5289.DBD156, 500 ms
   "2080SP241U01S01.Unit" : TextRef, internal   // Еденицы измерения При експорте из ECS через скрипт заполняется автоматически, если теги копируются в ручную то требуется задатать свойство Text
   "2080SP241U01S01.Decimals" : TextRef, internal   // Формат отображения При експорте из ECS через скрипт, заполняется автоматически. Если теги копируются в ручную то требуется задатать свойство Text s999999.9
   "2080SP241U01S01.FP_EN.Square" : Bool AT %DB5289.DBX46.0, 500 ms
   "2080SP241U01S01.FP_EN.SquareRoot" : Bool AT %DB5289.DBX46.1, 500 ms
   "2080SP241U01S01.FP_EN.ParentSupress" : Bool AT %DB5289.DBX46.2, 500 ms
   "2080SP241U01S01.FP_EN.ParentSupressUnit" : Bool AT %DB5289.DBX46.3, 500 ms
   "2080SP241U01S01.FP_EN.Force" : Bool AT %DB5289.DBX46.4, 500 ms
   "2080SP241U01S01.FP_EN.Damping" : Bool AT %DB5289.DBX46.5, 500 ms
   "2080SP241U01S01.FP_EN.Gradient_Pos" : Bool AT %DB5289.DBX46.6, 500 ms
   "2080SP241U01S01.FP_EN.Gradient_Neg" : Bool AT %DB5289.DBX46.7, 500 ms
   "2080SP241U01S01.FP_EN.Hysteresis" : Bool AT %DB5289.DBX47.0, 500 ms
   "2080SP241U01S01.FP_EN.Alarm_H3" : Bool AT %DB5289.DBX47.1, 500 ms
   "2080SP241U01S01.FP_EN.Alarm_H2" : Bool AT %DB5289.DBX47.2, 500 ms
   "2080SP241U01S01.FP_EN.Alarm_H1" : Bool AT %DB5289.DBX47.3, 500 ms
   "2080SP241U01S01.FP_EN.Alarm_L1" : Bool AT %DB5289.DBX47.4, 500 ms
   "2080SP241U01S01.FP_EN.Alarm_L2" : Bool AT %DB5289.DBX47.5, 500 ms
   "2080SP241U01S01.FP_EN.Alarm_L3" : Bool AT %DB5289.DBX47.6, 500 ms
   "2080SP241U01S01.FP_EN.AlarmDelay_H3" : Bool AT %DB5289.DBX47.7, 500 ms
   "2080SP241U01S01.FP_EN.AlarmDelay_H2" : Bool AT %DB5289.DBX48.0, 500 ms
   "2080SP241U01S01.FP_EN.AlarmDelay_H1" : Bool AT %DB5289.DBX48.1, 500 ms
   "2080SP241U01S01.FP_EN.AlarmDelay_L1" : Bool AT %DB5289.DBX48.2, 500 ms
   "2080SP241U01S01.FP_EN.AlarmDelay_L2" : Bool AT %DB5289.DBX48.3, 500 ms
   "2080SP241U01S01.FP_EN.AlarmDelay_L3" : Bool AT %DB5289.DBX48.4, 500 ms
   "2080SP241U01S01.FP_EN.ROC_Warn" : Bool AT %DB5289.DBX48.5, 500 ms
   "2080SP241U01S01.FP_EN.U_Range_Warn" : Bool AT %DB5289.DBX48.6, 500 ms
   "2080SP241U01S01.FP_EN.O_Range_Warn" : Bool AT %DB5289.DBX48.7, 500 ms
   "2080SP241U01S01.trend_tag_name" : TextRef, internal   // Еденицы измерения При експорте из ECS через скрипт - заполняется автоматически, если теги копируются в ручную то требуется задатать свойство Text - имя тега для тренда
   "2080SP241U01S01.DQ.AL_H3" : Bool AT %DB5289.DBX16.0, 500 ms
   "2080SP241U01S01.DQ.AL_H2" : Bool AT %DB5289.DBX16.1, 500 ms
   "2080SP241U01S01.DQ.AL_H1" : Bool AT %DB5289.DBX16.2, 500 ms
   "2080SP241U01S01.DQ.AL_L1" : Bool AT %DB5289.DBX16.3, 500 ms
   "2080SP241U01S01.DQ.AL_L2" : Bool AT %DB5289.DBX16.4, 500 ms
   "2080SP241U01S01.DQ.AL_L3" : Bool AT %DB5289.DBX16.5, 500 ms
   "2080SP241U01S01.DQ.SIG_OK" : Bool AT %DB5289.DBX16.6, 500 ms
   "2080SP241U01S01.DQ.LIM_H2" : Bool AT %DB5289.DBX16.7, 500 ms
   "2080SP241U01S01.DQ.LIM_H1" : Bool AT %DB5289.DBX17.0, 500 ms
   "2080SP241U01S01.DQ.LIM_L1" : Bool AT %DB5289.DBX17.1, 500 ms
   "2080SP241U01S01.DQ.LIM_L2" : Bool AT %DB5289.DBX17.2, 500 ms
   "2080SP241U01S01.DQ.GR_P" : Bool AT %DB5289.DBX17.3, 500 ms
   "2080SP241U01S01.DQ.GR_N" : Bool AT %DB5289.DBX17.4, 500 ms
   "2080SP241U01S01.I.IN" : Real AT %DB5289.DBD2, 500 ms
   "2080SP241U01S01.I.SIG_TYPE" : Int AT %DB5289.DBW0, 500 ms
   "2080SP241U01S01.I.FI_BUS" : Byte AT %DB5289.DBB6, 500 ms
   "2080SP241U01S01.DI.U_RANGE" : Bool AT %DB5289.DBX7.0, 500 ms
   "2080SP241U01S01.DI.O_RANGE" : Bool AT %DB5289.DBX7.1, 500 ms
   "2080SP241U01S01.DI.SIG_FAULT" : Bool AT %DB5289.DBX7.2, 500 ms
   "2080SP241U01S01.DI.EnConfig" : Bool AT %DB5289.DBX7.3, 500 ms
   "2080SP241U01S01.DI.AEN" : Bool AT %DB5289.DBX7.4, 500 ms
   "2080SP241U01S01.DI.AL_SUPR" : Bool AT %DB5289.DBX7.5, 500 ms
   "2080SP241U01S01.Q.PV_NORM" : Real AT %DB5289.DBD8, 500 ms
   "2080SP241U01S01.Q.PV_SCAL" : Real AT %DB5289.DBD12, 500 ms

HMI tags "2080TN450A01D01"
   "2080TN450A01D01.MSW" : 52809b66-421d-457f-8884-6f7a49d4e247 AT %DB5137.DBX18.0, 500 ms
   "2080TN450A01D01.DefaultText" : TextRef, internal   // Заголовок POPUP окна. При експорте из ECS через скрипт заполняется автоматически, если теги копируются в ручную то требуется в ручную задатать свойство Start Value
   "2080TN450A01D01.BlockInfo" : Array [0..2] of Int AT %DB5137.DBX38.0, 500 ms
   "2080TN450A01D01.StatusWork" : Int AT %DB5137.DBW242, 500 ms
   "2080TN450A01D01.FP_PARAM.DampingTime" : Int AT %DB5137.DBW50, 500 ms
   "2080TN450A01D01.FP_PARAM.Force_Value" : Real AT %DB5137.DBD52, 500 ms
   "2080TN450A01D01.FP_PARAM.Scale_Min" : Real AT %DB5137.DBD56, 500 ms
   "2080TN450A01D01.FP_PARAM.Scale_Max" : Real AT %DB5137.DBD60, 500 ms
   "2080TN450A01D01.FP_PARAM.Gradient" : Real AT %DB5137.DBD64, 500 ms
   "2080TN450A01D01.FP_PARAM.Grad_Pos" : Real AT %DB5137.DBD68, 500 ms
   "2080TN450A01D01.FP_PARAM.Grad_Neg" : Real AT %DB5137.DBD72, 500 ms
   "2080TN450A01D01.FP_PARAM.Grad_X" : Real AT %DB5137.DBD76, 500 ms
   "2080TN450A01D01.FP_PARAM.Gradient_Time_Pre" : Int AT %DB5137.DBW80, 500 ms
   "2080TN450A01D01.FP_PARAM.Gradient_Time_ACC" : Int AT %DB5137.DBW82, 500 ms
   "2080TN450A01D01.FP_PARAM.Alarm_Hyst" : Real AT %DB5137.DBD84, 500 ms
   "2080TN450A01D01.FP_PARAM.AlarmLimit_H3" : Real AT %DB5137.DBD88, 500 ms
   "2080TN450A01D01.FP_PARAM.AlarmLimit_H2" : Real AT %DB5137.DBD92, 500 ms
   "2080TN450A01D01.FP_PARAM.AlarmLimit_H1" : Real AT %DB5137.DBD96, 500 ms
   "2080TN450A01D01.FP_PARAM.AlarmLimit_L1" : Real AT %DB5137.DBD100, 500 ms
   "2080TN450A01D01.FP_PARAM.AlarmLimit_L2" : Real AT %DB5137.DBD104, 500 ms
   "2080TN450A01D01.FP_PARAM.AlarmLimit_L3" : Real AT %DB5137.DBD108, 500 ms
   "2080TN450A01D01.FP_PARAM.AlarmDelay_H3_Pre" : Int AT %DB5137.DBW112, 500 ms
   "2080TN450A01D01.FP_PARAM.AlarmDelay_H3_Acc" : Int AT %DB5137.DBW114, 500 ms
   "2080TN450A01D01.FP_PARAM.AlarmDelay_H2_Pre" : Int AT %DB5137.DBW116, 500 ms
   "2080TN450A01D01.FP_PARAM.AlarmDelay_H2_Acc" : Int AT %DB5137.DBW118, 500 ms
   "2080TN450A01D01.FP_PARAM.AlarmDelay_H1_Pre" : Int AT %DB5137.DBW120, 500 ms
   "2080TN450A01D01.FP_PARAM.AlarmDelay_H1_Acc" : Int AT %DB5137.DBW122, 500 ms
   "2080TN450A01D01.FP_PARAM.AlarmDelay_L1_Pre" : Int AT %DB5137.DBW124, 500 ms
   "2080TN450A01D01.FP_PARAM.AlarmDelay_L1_Acc" : Int AT %DB5137.DBW126, 500 ms
   "2080TN450A01D01.FP_PARAM.AlarmDelay_L2_Pre" : Int AT %DB5137.DBW128, 500 ms
   "2080TN450A01D01.FP_PARAM.AlarmDelay_L2_Acc" : Int AT %DB5137.DBW130, 500 ms
   "2080TN450A01D01.FP_PARAM.AlarmDelay_L3_Pre" : Int AT %DB5137.DBW132, 500 ms
   "2080TN450A01D01.FP_PARAM.AlarmDelay_L3_Acc" : Int AT %DB5137.DBW134, 500 ms
   "2080TN450A01D01.FP_PARAM.OpenLoopDelay_Pre" : Int AT %DB5137.DBW136, 500 ms
   "2080TN450A01D01.FP_PARAM.OpenLoopDelay_Acc" : Int AT %DB5137.DBW138, 500 ms
   "2080TN450A01D01.FP_PARAM.OverRangeDelay_Pre" : Int AT %DB5137.DBW140, 500 ms
   "2080TN450A01D01.FP_PARAM.OverRangeDelay_Acc" : Int AT %DB5137.DBW142, 500 ms
   "2080TN450A01D01.FP_PARAM.AuxLimit_H2_Value" : Real AT %DB5137.DBD144, 500 ms
   "2080TN450A01D01.FP_PARAM.AuxLimit_H1_Value" : Real AT %DB5137.DBD148, 500 ms
   "2080TN450A01D01.FP_PARAM.AuxLimit_L2_Value" : Real AT %DB5137.DBD152, 500 ms
   "2080TN450A01D01.FP_PARAM.AuxLimit_L1_Value" : Real AT %DB5137.DBD156, 500 ms
   "2080TN450A01D01.Unit" : TextRef, internal   // Еденицы измерения При експорте из ECS через скрипт заполняется автоматически, если теги копируются в ручную то требуется задатать свойство Text
   "2080TN450A01D01.Decimals" : TextRef, internal   // Формат отображения При експорте из ECS через скрипт, заполняется автоматически. Если теги копируются в ручную то требуется задатать свойство Text s999999.9
   "2080TN450A01D01.FP_EN.Square" : Bool AT %DB5137.DBX46.0, 500 ms
   "2080TN450A01D01.FP_EN.SquareRoot" : Bool AT %DB5137.DBX46.1, 500 ms
   "2080TN450A01D01.FP_EN.ParentSupress" : Bool AT %DB5137.DBX46.2, 500 ms
   "2080TN450A01D01.FP_EN.ParentSupressUnit" : Bool AT %DB5137.DBX46.3, 500 ms
   "2080TN450A01D01.FP_EN.Force" : Bool AT %DB5137.DBX46.4, 500 ms
   "2080TN450A01D01.FP_EN.Damping" : Bool AT %DB5137.DBX46.5, 500 ms
   "2080TN450A01D01.FP_EN.Gradient_Pos" : Bool AT %DB5137.DBX46.6, 500 ms
   "2080TN450A01D01.FP_EN.Gradient_Neg" : Bool AT %DB5137.DBX46.7, 500 ms
   "2080TN450A01D01.FP_EN.Hysteresis" : Bool AT %DB5137.DBX47.0, 500 ms
   "2080TN450A01D01.FP_EN.Alarm_H3" : Bool AT %DB5137.DBX47.1, 500 ms
   "2080TN450A01D01.FP_EN.Alarm_H2" : Bool AT %DB5137.DBX47.2, 500 ms
   "2080TN450A01D01.FP_EN.Alarm_H1" : Bool AT %DB5137.DBX47.3, 500 ms
   "2080TN450A01D01.FP_EN.Alarm_L1" : Bool AT %DB5137.DBX47.4, 500 ms
   "2080TN450A01D01.FP_EN.Alarm_L2" : Bool AT %DB5137.DBX47.5, 500 ms
   "2080TN450A01D01.FP_EN.Alarm_L3" : Bool AT %DB5137.DBX47.6, 500 ms
   "2080TN450A01D01.FP_EN.AlarmDelay_H3" : Bool AT %DB5137.DBX47.7, 500 ms
   "2080TN450A01D01.FP_EN.AlarmDelay_H2" : Bool AT %DB5137.DBX48.0, 500 ms
   "2080TN450A01D01.FP_EN.AlarmDelay_H1" : Bool AT %DB5137.DBX48.1, 500 ms
   "2080TN450A01D01.FP_EN.AlarmDelay_L1" : Bool AT %DB5137.DBX48.2, 500 ms
   "2080TN450A01D01.FP_EN.AlarmDelay_L2" : Bool AT %DB5137.DBX48.3, 500 ms
   "2080TN450A01D01.FP_EN.AlarmDelay_L3" : Bool AT %DB5137.DBX48.4, 500 ms
   "2080TN450A01D01.FP_EN.ROC_Warn" : Bool AT %DB5137.DBX48.5, 500 ms
   "2080TN450A01D01.FP_EN.U_Range_Warn" : Bool AT %DB5137.DBX48.6, 500 ms
   "2080TN450A01D01.FP_EN.O_Range_Warn" : Bool AT %DB5137.DBX48.7, 500 ms
   "2080TN450A01D01.trend_tag_name" : TextRef, internal   // Еденицы измерения При експорте из ECS через скрипт - заполняется автоматически, если теги копируются в ручную то требуется задатать свойство Text - имя тега для тренда
   "2080TN450A01D01.DQ.AL_H3" : Bool AT %DB5137.DBX16.0, 500 ms
   "2080TN450A01D01.DQ.AL_H2" : Bool AT %DB5137.DBX16.1, 500 ms
   "2080TN450A01D01.DQ.AL_H1" : Bool AT %DB5137.DBX16.2, 500 ms
   "2080TN450A01D01.DQ.AL_L1" : Bool AT %DB5137.DBX16.3, 500 ms
   "2080TN450A01D01.DQ.AL_L2" : Bool AT %DB5137.DBX16.4, 500 ms
   "2080TN450A01D01.DQ.AL_L3" : Bool AT %DB5137.DBX16.5, 500 ms
   "2080TN450A01D01.DQ.SIG_OK" : Bool AT %DB5137.DBX16.6, 500 ms
   "2080TN450A01D01.DQ.LIM_H2" : Bool AT %DB5137.DBX16.7, 500 ms
   "2080TN450A01D01.DQ.LIM_H1" : Bool AT %DB5137.DBX17.0, 500 ms
   "2080TN450A01D01.DQ.LIM_L1" : Bool AT %DB5137.DBX17.1, 500 ms
   "2080TN450A01D01.DQ.LIM_L2" : Bool AT %DB5137.DBX17.2, 500 ms
   "2080TN450A01D01.DQ.GR_P" : Bool AT %DB5137.DBX17.3, 500 ms
   "2080TN450A01D01.DQ.GR_N" : Bool AT %DB5137.DBX17.4, 500 ms
   "2080TN450A01D01.I.IN" : Real AT %DB5137.DBD2, 500 ms
   "2080TN450A01D01.I.SIG_TYPE" : Int AT %DB5137.DBW0, 500 ms
   "2080TN450A01D01.I.FI_BUS" : Byte AT %DB5137.DBB6, 500 ms
   "2080TN450A01D01.DI.U_RANGE" : Bool AT %DB5137.DBX7.0, 500 ms
   "2080TN450A01D01.DI.O_RANGE" : Bool AT %DB5137.DBX7.1, 500 ms
   "2080TN450A01D01.DI.SIG_FAULT" : Bool AT %DB5137.DBX7.2, 500 ms
   "2080TN450A01D01.DI.EnConfig" : Bool AT %DB5137.DBX7.3, 500 ms
   "2080TN450A01D01.DI.AEN" : Bool AT %DB5137.DBX7.4, 500 ms
   "2080TN450A01D01.DI.AL_SUPR" : Bool AT %DB5137.DBX7.5, 500 ms
   "2080TN450A01D01.Q.PV_NORM" : Real AT %DB5137.DBD8, 500 ms
   "2080TN450A01D01.Q.PV_SCAL" : Real AT %DB5137.DBD12, 500 ms
   "2080TN450A01D01.ParentInfo" : TextRef, internal   // Имя родителя для попап окна, вкладка инфо. При експорте из ECS через скрипт заполняется автоматически, если теги копируются в ручную то требуется в ручную задатать свойство Start Value

HMI tags "2080TN450A01F01"
   "2080TN450A01F01.MSW" : 52809b66-421d-457f-8884-6f7a49d4e247 AT %DB5138.DBX18.0, 500 ms
   "2080TN450A01F01.DefaultText" : TextRef, internal   // Заголовок POPUP окна. При експорте из ECS через скрипт заполняется автоматически, если теги копируются в ручную то требуется в ручную задатать свойство Start Value
   "2080TN450A01F01.BlockInfo" : Array [0..2] of Int AT %DB5138.DBX38.0, 500 ms
   "2080TN450A01F01.StatusWork" : Int AT %DB5138.DBW242, 500 ms
   "2080TN450A01F01.FP_PARAM.DampingTime" : Int AT %DB5138.DBW50, 500 ms
   "2080TN450A01F01.FP_PARAM.Force_Value" : Real AT %DB5138.DBD52, 500 ms
   "2080TN450A01F01.FP_PARAM.Scale_Min" : Real AT %DB5138.DBD56, 500 ms
   "2080TN450A01F01.FP_PARAM.Scale_Max" : Real AT %DB5138.DBD60, 500 ms
   "2080TN450A01F01.FP_PARAM.Gradient" : Real AT %DB5138.DBD64, 500 ms
   "2080TN450A01F01.FP_PARAM.Grad_Pos" : Real AT %DB5138.DBD68, 500 ms
   "2080TN450A01F01.FP_PARAM.Grad_Neg" : Real AT %DB5138.DBD72, 500 ms
   "2080TN450A01F01.FP_PARAM.Grad_X" : Real AT %DB5138.DBD76, 500 ms
   "2080TN450A01F01.FP_PARAM.Gradient_Time_Pre" : Int AT %DB5138.DBW80, 500 ms
   "2080TN450A01F01.FP_PARAM.Gradient_Time_ACC" : Int AT %DB5138.DBW82, 500 ms
   "2080TN450A01F01.FP_PARAM.Alarm_Hyst" : Real AT %DB5138.DBD84, 500 ms
   "2080TN450A01F01.FP_PARAM.AlarmLimit_H3" : Real AT %DB5138.DBD88, 500 ms
   "2080TN450A01F01.FP_PARAM.AlarmLimit_H2" : Real AT %DB5138.DBD92, 500 ms
   "2080TN450A01F01.FP_PARAM.AlarmLimit_H1" : Real AT %DB5138.DBD96, 500 ms
   "2080TN450A01F01.FP_PARAM.AlarmLimit_L1" : Real AT %DB5138.DBD100, 500 ms
   "2080TN450A01F01.FP_PARAM.AlarmLimit_L2" : Real AT %DB5138.DBD104, 500 ms
   "2080TN450A01F01.FP_PARAM.AlarmLimit_L3" : Real AT %DB5138.DBD108, 500 ms
   "2080TN450A01F01.FP_PARAM.AlarmDelay_H3_Pre" : Int AT %DB5138.DBW112, 500 ms
   "2080TN450A01F01.FP_PARAM.AlarmDelay_H3_Acc" : Int AT %DB5138.DBW114, 500 ms
   "2080TN450A01F01.FP_PARAM.AlarmDelay_H2_Pre" : Int AT %DB5138.DBW116, 500 ms
   "2080TN450A01F01.FP_PARAM.AlarmDelay_H2_Acc" : Int AT %DB5138.DBW118, 500 ms
   "2080TN450A01F01.FP_PARAM.AlarmDelay_H1_Pre" : Int AT %DB5138.DBW120, 500 ms
   "2080TN450A01F01.FP_PARAM.AlarmDelay_H1_Acc" : Int AT %DB5138.DBW122, 500 ms
   "2080TN450A01F01.FP_PARAM.AlarmDelay_L1_Pre" : Int AT %DB5138.DBW124, 500 ms
   "2080TN450A01F01.FP_PARAM.AlarmDelay_L1_Acc" : Int AT %DB5138.DBW126, 500 ms
   "2080TN450A01F01.FP_PARAM.AlarmDelay_L2_Pre" : Int AT %DB5138.DBW128, 500 ms
   "2080TN450A01F01.FP_PARAM.AlarmDelay_L2_Acc" : Int AT %DB5138.DBW130, 500 ms
   "2080TN450A01F01.FP_PARAM.AlarmDelay_L3_Pre" : Int AT %DB5138.DBW132, 500 ms
   "2080TN450A01F01.FP_PARAM.AlarmDelay_L3_Acc" : Int AT %DB5138.DBW134, 500 ms
   "2080TN450A01F01.FP_PARAM.OpenLoopDelay_Pre" : Int AT %DB5138.DBW136, 500 ms
   "2080TN450A01F01.FP_PARAM.OpenLoopDelay_Acc" : Int AT %DB5138.DBW138, 500 ms
   "2080TN450A01F01.FP_PARAM.OverRangeDelay_Pre" : Int AT %DB5138.DBW140, 500 ms
   "2080TN450A01F01.FP_PARAM.OverRangeDelay_Acc" : Int AT %DB5138.DBW142, 500 ms
   "2080TN450A01F01.FP_PARAM.AuxLimit_H2_Value" : Real AT %DB5138.DBD144, 500 ms
   "2080TN450A01F01.FP_PARAM.AuxLimit_H1_Value" : Real AT %DB5138.DBD148, 500 ms
   "2080TN450A01F01.FP_PARAM.AuxLimit_L2_Value" : Real AT %DB5138.DBD152, 500 ms
   "2080TN450A01F01.FP_PARAM.AuxLimit_L1_Value" : Real AT %DB5138.DBD156, 500 ms
   "2080TN450A01F01.Unit" : TextRef, internal   // Еденицы измерения При експорте из ECS через скрипт заполняется автоматически, если теги копируются в ручную то требуется задатать свойство Text
   "2080TN450A01F01.Decimals" : TextRef, internal   // Формат отображения При експорте из ECS через скрипт, заполняется автоматически. Если теги копируются в ручную то требуется задатать свойство Text s999999.9
   "2080TN450A01F01.FP_EN.Square" : Bool AT %DB5138.DBX46.0, 500 ms
   "2080TN450A01F01.FP_EN.SquareRoot" : Bool AT %DB5138.DBX46.1, 500 ms
   "2080TN450A01F01.FP_EN.ParentSupress" : Bool AT %DB5138.DBX46.2, 500 ms
   "2080TN450A01F01.FP_EN.ParentSupressUnit" : Bool AT %DB5138.DBX46.3, 500 ms
   "2080TN450A01F01.FP_EN.Force" : Bool AT %DB5138.DBX46.4, 500 ms
   "2080TN450A01F01.FP_EN.Damping" : Bool AT %DB5138.DBX46.5, 500 ms
   "2080TN450A01F01.FP_EN.Gradient_Pos" : Bool AT %DB5138.DBX46.6, 500 ms
   "2080TN450A01F01.FP_EN.Gradient_Neg" : Bool AT %DB5138.DBX46.7, 500 ms
   "2080TN450A01F01.FP_EN.Hysteresis" : Bool AT %DB5138.DBX47.0, 500 ms
   "2080TN450A01F01.FP_EN.Alarm_H3" : Bool AT %DB5138.DBX47.1, 500 ms
   "2080TN450A01F01.FP_EN.Alarm_H2" : Bool AT %DB5138.DBX47.2, 500 ms
   "2080TN450A01F01.FP_EN.Alarm_H1" : Bool AT %DB5138.DBX47.3, 500 ms
   "2080TN450A01F01.FP_EN.Alarm_L1" : Bool AT %DB5138.DBX47.4, 500 ms
   "2080TN450A01F01.FP_EN.Alarm_L2" : Bool AT %DB5138.DBX47.5, 500 ms
   "2080TN450A01F01.FP_EN.Alarm_L3" : Bool AT %DB5138.DBX47.6, 500 ms
   "2080TN450A01F01.FP_EN.AlarmDelay_H3" : Bool AT %DB5138.DBX47.7, 500 ms
   "2080TN450A01F01.FP_EN.AlarmDelay_H2" : Bool AT %DB5138.DBX48.0, 500 ms
   "2080TN450A01F01.FP_EN.AlarmDelay_H1" : Bool AT %DB5138.DBX48.1, 500 ms
   "2080TN450A01F01.FP_EN.AlarmDelay_L1" : Bool AT %DB5138.DBX48.2, 500 ms
   "2080TN450A01F01.FP_EN.AlarmDelay_L2" : Bool AT %DB5138.DBX48.3, 500 ms
   "2080TN450A01F01.FP_EN.AlarmDelay_L3" : Bool AT %DB5138.DBX48.4, 500 ms
   "2080TN450A01F01.FP_EN.ROC_Warn" : Bool AT %DB5138.DBX48.5, 500 ms
   "2080TN450A01F01.FP_EN.U_Range_Warn" : Bool AT %DB5138.DBX48.6, 500 ms
   "2080TN450A01F01.FP_EN.O_Range_Warn" : Bool AT %DB5138.DBX48.7, 500 ms
   "2080TN450A01F01.trend_tag_name" : TextRef, internal   // Еденицы измерения При експорте из ECS через скрипт - заполняется автоматически, если теги копируются в ручную то требуется задатать свойство Text - имя тега для тренда
   "2080TN450A01F01.DQ.AL_H3" : Bool AT %DB5138.DBX16.0, 500 ms
   "2080TN450A01F01.DQ.AL_H2" : Bool AT %DB5138.DBX16.1, 500 ms
   "2080TN450A01F01.DQ.AL_H1" : Bool AT %DB5138.DBX16.2, 500 ms
   "2080TN450A01F01.DQ.AL_L1" : Bool AT %DB5138.DBX16.3, 500 ms
   "2080TN450A01F01.DQ.AL_L2" : Bool AT %DB5138.DBX16.4, 500 ms
   "2080TN450A01F01.DQ.AL_L3" : Bool AT %DB5138.DBX16.5, 500 ms
   "2080TN450A01F01.DQ.SIG_OK" : Bool AT %DB5138.DBX16.6, 500 ms
   "2080TN450A01F01.DQ.LIM_H2" : Bool AT %DB5138.DBX16.7, 500 ms
   "2080TN450A01F01.DQ.LIM_H1" : Bool AT %DB5138.DBX17.0, 500 ms
   "2080TN450A01F01.DQ.LIM_L1" : Bool AT %DB5138.DBX17.1, 500 ms
   "2080TN450A01F01.DQ.LIM_L2" : Bool AT %DB5138.DBX17.2, 500 ms
   "2080TN450A01F01.DQ.GR_P" : Bool AT %DB5138.DBX17.3, 500 ms
   "2080TN450A01F01.DQ.GR_N" : Bool AT %DB5138.DBX17.4, 500 ms
   "2080TN450A01F01.I.IN" : Real AT %DB5138.DBD2, 500 ms
   "2080TN450A01F01.I.SIG_TYPE" : Int AT %DB5138.DBW0, 500 ms
   "2080TN450A01F01.I.FI_BUS" : Byte AT %DB5138.DBB6, 500 ms
   "2080TN450A01F01.DI.U_RANGE" : Bool AT %DB5138.DBX7.0, 500 ms
   "2080TN450A01F01.DI.O_RANGE" : Bool AT %DB5138.DBX7.1, 500 ms
   "2080TN450A01F01.DI.SIG_FAULT" : Bool AT %DB5138.DBX7.2, 500 ms
   "2080TN450A01F01.DI.EnConfig" : Bool AT %DB5138.DBX7.3, 500 ms
   "2080TN450A01F01.DI.AEN" : Bool AT %DB5138.DBX7.4, 500 ms
   "2080TN450A01F01.DI.AL_SUPR" : Bool AT %DB5138.DBX7.5, 500 ms
   "2080TN450A01F01.Q.PV_NORM" : Real AT %DB5138.DBD8, 500 ms
   "2080TN450A01F01.Q.PV_SCAL" : Real AT %DB5138.DBD12, 500 ms
   "2080TN450A01F01.ParentInfo" : TextRef, internal   // Имя родителя для попап окна, вкладка инфо. При експорте из ECS через скрипт заполняется автоматически, если теги копируются в ручную то требуется в ручную задатать свойство Start Value

HMI tags "2080TN450A01I01"
   "2080TN450A01I01.MSW" : 52809b66-421d-457f-8884-6f7a49d4e247 AT %DB5123.DBX18.0, 500 ms
   "2080TN450A01I01.DefaultText" : TextRef, internal   // Заголовок POPUP окна. При експорте из ECS через скрипт заполняется автоматически, если теги копируются в ручную то требуется в ручную задатать свойство Start Value
   "2080TN450A01I01.BlockInfo" : Array [0..2] of Int AT %DB5123.DBX38.0, 500 ms
   "2080TN450A01I01.StatusWork" : Int AT %DB5123.DBW242, 500 ms
   "2080TN450A01I01.FP_PARAM.DampingTime" : Int AT %DB5123.DBW50, 500 ms
   "2080TN450A01I01.FP_PARAM.Force_Value" : Real AT %DB5123.DBD52, 500 ms
   "2080TN450A01I01.FP_PARAM.Scale_Min" : Real AT %DB5123.DBD56, 500 ms
   "2080TN450A01I01.FP_PARAM.Scale_Max" : Real AT %DB5123.DBD60, 500 ms
   "2080TN450A01I01.FP_PARAM.Gradient" : Real AT %DB5123.DBD64, 500 ms
   "2080TN450A01I01.FP_PARAM.Grad_Pos" : Real AT %DB5123.DBD68, 500 ms
   "2080TN450A01I01.FP_PARAM.Grad_Neg" : Real AT %DB5123.DBD72, 500 ms
   "2080TN450A01I01.FP_PARAM.Grad_X" : Real AT %DB5123.DBD76, 500 ms
   "2080TN450A01I01.FP_PARAM.Gradient_Time_Pre" : Int AT %DB5123.DBW80, 500 ms
   "2080TN450A01I01.FP_PARAM.Gradient_Time_ACC" : Int AT %DB5123.DBW82, 500 ms
   "2080TN450A01I01.FP_PARAM.Alarm_Hyst" : Real AT %DB5123.DBD84, 500 ms
   "2080TN450A01I01.FP_PARAM.AlarmLimit_H3" : Real AT %DB5123.DBD88, 500 ms
   "2080TN450A01I01.FP_PARAM.AlarmLimit_H2" : Real AT %DB5123.DBD92, 500 ms
   "2080TN450A01I01.FP_PARAM.AlarmLimit_H1" : Real AT %DB5123.DBD96, 500 ms
   "2080TN450A01I01.FP_PARAM.AlarmLimit_L1" : Real AT %DB5123.DBD100, 500 ms
   "2080TN450A01I01.FP_PARAM.AlarmLimit_L2" : Real AT %DB5123.DBD104, 500 ms
   "2080TN450A01I01.FP_PARAM.AlarmLimit_L3" : Real AT %DB5123.DBD108, 500 ms
   "2080TN450A01I01.FP_PARAM.AlarmDelay_H3_Pre" : Int AT %DB5123.DBW112, 500 ms
   "2080TN450A01I01.FP_PARAM.AlarmDelay_H3_Acc" : Int AT %DB5123.DBW114, 500 ms
   "2080TN450A01I01.FP_PARAM.AlarmDelay_H2_Pre" : Int AT %DB5123.DBW116, 500 ms
   "2080TN450A01I01.FP_PARAM.AlarmDelay_H2_Acc" : Int AT %DB5123.DBW118, 500 ms
   "2080TN450A01I01.FP_PARAM.AlarmDelay_H1_Pre" : Int AT %DB5123.DBW120, 500 ms
   "2080TN450A01I01.FP_PARAM.AlarmDelay_H1_Acc" : Int AT %DB5123.DBW122, 500 ms
   "2080TN450A01I01.FP_PARAM.AlarmDelay_L1_Pre" : Int AT %DB5123.DBW124, 500 ms
   "2080TN450A01I01.FP_PARAM.AlarmDelay_L1_Acc" : Int AT %DB5123.DBW126, 500 ms
   "2080TN450A01I01.FP_PARAM.AlarmDelay_L2_Pre" : Int AT %DB5123.DBW128, 500 ms
   "2080TN450A01I01.FP_PARAM.AlarmDelay_L2_Acc" : Int AT %DB5123.DBW130, 500 ms
   "2080TN450A01I01.FP_PARAM.AlarmDelay_L3_Pre" : Int AT %DB5123.DBW132, 500 ms
   "2080TN450A01I01.FP_PARAM.AlarmDelay_L3_Acc" : Int AT %DB5123.DBW134, 500 ms
   "2080TN450A01I01.FP_PARAM.OpenLoopDelay_Pre" : Int AT %DB5123.DBW136, 500 ms
   "2080TN450A01I01.FP_PARAM.OpenLoopDelay_Acc" : Int AT %DB5123.DBW138, 500 ms
   "2080TN450A01I01.FP_PARAM.OverRangeDelay_Pre" : Int AT %DB5123.DBW140, 500 ms
   "2080TN450A01I01.FP_PARAM.OverRangeDelay_Acc" : Int AT %DB5123.DBW142, 500 ms
   "2080TN450A01I01.FP_PARAM.AuxLimit_H2_Value" : Real AT %DB5123.DBD144, 500 ms
   "2080TN450A01I01.FP_PARAM.AuxLimit_H1_Value" : Real AT %DB5123.DBD148, 500 ms
   "2080TN450A01I01.FP_PARAM.AuxLimit_L2_Value" : Real AT %DB5123.DBD152, 500 ms
   "2080TN450A01I01.FP_PARAM.AuxLimit_L1_Value" : Real AT %DB5123.DBD156, 500 ms
   "2080TN450A01I01.Unit" : TextRef, internal   // Еденицы измерения При експорте из ECS через скрипт заполняется автоматически, если теги копируются в ручную то требуется задатать свойство Text
   "2080TN450A01I01.Decimals" : TextRef, internal   // Формат отображения При експорте из ECS через скрипт, заполняется автоматически. Если теги копируются в ручную то требуется задатать свойство Text s999999.9
   "2080TN450A01I01.FP_EN.Square" : Bool AT %DB5123.DBX46.0, 500 ms
   "2080TN450A01I01.FP_EN.SquareRoot" : Bool AT %DB5123.DBX46.1, 500 ms
   "2080TN450A01I01.FP_EN.ParentSupress" : Bool AT %DB5123.DBX46.2, 500 ms
   "2080TN450A01I01.FP_EN.ParentSupressUnit" : Bool AT %DB5123.DBX46.3, 500 ms
   "2080TN450A01I01.FP_EN.Force" : Bool AT %DB5123.DBX46.4, 500 ms
   "2080TN450A01I01.FP_EN.Damping" : Bool AT %DB5123.DBX46.5, 500 ms
   "2080TN450A01I01.FP_EN.Gradient_Pos" : Bool AT %DB5123.DBX46.6, 500 ms
   "2080TN450A01I01.FP_EN.Gradient_Neg" : Bool AT %DB5123.DBX46.7, 500 ms
   "2080TN450A01I01.FP_EN.Hysteresis" : Bool AT %DB5123.DBX47.0, 500 ms
   "2080TN450A01I01.FP_EN.Alarm_H3" : Bool AT %DB5123.DBX47.1, 500 ms
   "2080TN450A01I01.FP_EN.Alarm_H2" : Bool AT %DB5123.DBX47.2, 500 ms
   "2080TN450A01I01.FP_EN.Alarm_H1" : Bool AT %DB5123.DBX47.3, 500 ms
   "2080TN450A01I01.FP_EN.Alarm_L1" : Bool AT %DB5123.DBX47.4, 500 ms
   "2080TN450A01I01.FP_EN.Alarm_L2" : Bool AT %DB5123.DBX47.5, 500 ms
   "2080TN450A01I01.FP_EN.Alarm_L3" : Bool AT %DB5123.DBX47.6, 500 ms
   "2080TN450A01I01.FP_EN.AlarmDelay_H3" : Bool AT %DB5123.DBX47.7, 500 ms
   "2080TN450A01I01.FP_EN.AlarmDelay_H2" : Bool AT %DB5123.DBX48.0, 500 ms
   "2080TN450A01I01.FP_EN.AlarmDelay_H1" : Bool AT %DB5123.DBX48.1, 500 ms
   "2080TN450A01I01.FP_EN.AlarmDelay_L1" : Bool AT %DB5123.DBX48.2, 500 ms
   "2080TN450A01I01.FP_EN.AlarmDelay_L2" : Bool AT %DB5123.DBX48.3, 500 ms
   "2080TN450A01I01.FP_EN.AlarmDelay_L3" : Bool AT %DB5123.DBX48.4, 500 ms
   "2080TN450A01I01.FP_EN.ROC_Warn" : Bool AT %DB5123.DBX48.5, 500 ms
   "2080TN450A01I01.FP_EN.U_Range_Warn" : Bool AT %DB5123.DBX48.6, 500 ms
   "2080TN450A01I01.FP_EN.O_Range_Warn" : Bool AT %DB5123.DBX48.7, 500 ms
   "2080TN450A01I01.trend_tag_name" : TextRef, internal   // Еденицы измерения При експорте из ECS через скрипт - заполняется автоматически, если теги копируются в ручную то требуется задатать свойство Text - имя тега для тренда
   "2080TN450A01I01.DQ.AL_H3" : Bool AT %DB5123.DBX16.0, 500 ms
   "2080TN450A01I01.DQ.AL_H2" : Bool AT %DB5123.DBX16.1, 500 ms
   "2080TN450A01I01.DQ.AL_H1" : Bool AT %DB5123.DBX16.2, 500 ms
   "2080TN450A01I01.DQ.AL_L1" : Bool AT %DB5123.DBX16.3, 500 ms
   "2080TN450A01I01.DQ.AL_L2" : Bool AT %DB5123.DBX16.4, 500 ms
   "2080TN450A01I01.DQ.AL_L3" : Bool AT %DB5123.DBX16.5, 500 ms
   "2080TN450A01I01.DQ.SIG_OK" : Bool AT %DB5123.DBX16.6, 500 ms
   "2080TN450A01I01.DQ.LIM_H2" : Bool AT %DB5123.DBX16.7, 500 ms
   "2080TN450A01I01.DQ.LIM_H1" : Bool AT %DB5123.DBX17.0, 500 ms
   "2080TN450A01I01.DQ.LIM_L1" : Bool AT %DB5123.DBX17.1, 500 ms
   "2080TN450A01I01.DQ.LIM_L2" : Bool AT %DB5123.DBX17.2, 500 ms
   "2080TN450A01I01.DQ.GR_P" : Bool AT %DB5123.DBX17.3, 500 ms
   "2080TN450A01I01.DQ.GR_N" : Bool AT %DB5123.DBX17.4, 500 ms
   "2080TN450A01I01.I.IN" : Real AT %DB5123.DBD2, 500 ms
   "2080TN450A01I01.I.SIG_TYPE" : Int AT %DB5123.DBW0, 500 ms
   "2080TN450A01I01.I.FI_BUS" : Byte AT %DB5123.DBB6, 500 ms
   "2080TN450A01I01.DI.U_RANGE" : Bool AT %DB5123.DBX7.0, 500 ms
   "2080TN450A01I01.DI.O_RANGE" : Bool AT %DB5123.DBX7.1, 500 ms
   "2080TN450A01I01.DI.SIG_FAULT" : Bool AT %DB5123.DBX7.2, 500 ms
   "2080TN450A01I01.DI.EnConfig" : Bool AT %DB5123.DBX7.3, 500 ms
   "2080TN450A01I01.DI.AEN" : Bool AT %DB5123.DBX7.4, 500 ms
   "2080TN450A01I01.DI.AL_SUPR" : Bool AT %DB5123.DBX7.5, 500 ms
   "2080TN450A01I01.Q.PV_NORM" : Real AT %DB5123.DBD8, 500 ms
   "2080TN450A01I01.Q.PV_SCAL" : Real AT %DB5123.DBD12, 500 ms
   "2080TN450A01I01.ParentInfo" : TextRef, internal   // Имя родителя для попап окна, вкладка инфо. При експорте из ECS через скрипт заполняется автоматически, если теги копируются в ручную то требуется в ручную задатать свойство Start Value

HMI tags "2080TN450A01I02"
   "2080TN450A01I02.MSW" : 52809b66-421d-457f-8884-6f7a49d4e247 AT %DB5124.DBX18.0, 500 ms
   "2080TN450A01I02.DefaultText" : TextRef, internal   // Заголовок POPUP окна. При експорте из ECS через скрипт заполняется автоматически, если теги копируются в ручную то требуется в ручную задатать свойство Start Value
   "2080TN450A01I02.BlockInfo" : Array [0..2] of Int AT %DB5124.DBX38.0, 500 ms
   "2080TN450A01I02.StatusWork" : Int AT %DB5124.DBW242, 500 ms
   "2080TN450A01I02.FP_PARAM.DampingTime" : Int AT %DB5124.DBW50, 500 ms
   "2080TN450A01I02.FP_PARAM.Force_Value" : Real AT %DB5124.DBD52, 500 ms
   "2080TN450A01I02.FP_PARAM.Scale_Min" : Real AT %DB5124.DBD56, 500 ms
   "2080TN450A01I02.FP_PARAM.Scale_Max" : Real AT %DB5124.DBD60, 500 ms
   "2080TN450A01I02.FP_PARAM.Gradient" : Real AT %DB5124.DBD64, 500 ms
   "2080TN450A01I02.FP_PARAM.Grad_Pos" : Real AT %DB5124.DBD68, 500 ms
   "2080TN450A01I02.FP_PARAM.Grad_Neg" : Real AT %DB5124.DBD72, 500 ms
   "2080TN450A01I02.FP_PARAM.Grad_X" : Real AT %DB5124.DBD76, 500 ms
   "2080TN450A01I02.FP_PARAM.Gradient_Time_Pre" : Int AT %DB5124.DBW80, 500 ms
   "2080TN450A01I02.FP_PARAM.Gradient_Time_ACC" : Int AT %DB5124.DBW82, 500 ms
   "2080TN450A01I02.FP_PARAM.Alarm_Hyst" : Real AT %DB5124.DBD84, 500 ms
   "2080TN450A01I02.FP_PARAM.AlarmLimit_H3" : Real AT %DB5124.DBD88, 500 ms
   "2080TN450A01I02.FP_PARAM.AlarmLimit_H2" : Real AT %DB5124.DBD92, 500 ms
   "2080TN450A01I02.FP_PARAM.AlarmLimit_H1" : Real AT %DB5124.DBD96, 500 ms
   "2080TN450A01I02.FP_PARAM.AlarmLimit_L1" : Real AT %DB5124.DBD100, 500 ms
   "2080TN450A01I02.FP_PARAM.AlarmLimit_L2" : Real AT %DB5124.DBD104, 500 ms
   "2080TN450A01I02.FP_PARAM.AlarmLimit_L3" : Real AT %DB5124.DBD108, 500 ms
   "2080TN450A01I02.FP_PARAM.AlarmDelay_H3_Pre" : Int AT %DB5124.DBW112, 500 ms
   "2080TN450A01I02.FP_PARAM.AlarmDelay_H3_Acc" : Int AT %DB5124.DBW114, 500 ms
   "2080TN450A01I02.FP_PARAM.AlarmDelay_H2_Pre" : Int AT %DB5124.DBW116, 500 ms
   "2080TN450A01I02.FP_PARAM.AlarmDelay_H2_Acc" : Int AT %DB5124.DBW118, 500 ms
   "2080TN450A01I02.FP_PARAM.AlarmDelay_H1_Pre" : Int AT %DB5124.DBW120, 500 ms
   "2080TN450A01I02.FP_PARAM.AlarmDelay_H1_Acc" : Int AT %DB5124.DBW122, 500 ms
   "2080TN450A01I02.FP_PARAM.AlarmDelay_L1_Pre" : Int AT %DB5124.DBW124, 500 ms
   "2080TN450A01I02.FP_PARAM.AlarmDelay_L1_Acc" : Int AT %DB5124.DBW126, 500 ms
   "2080TN450A01I02.FP_PARAM.AlarmDelay_L2_Pre" : Int AT %DB5124.DBW128, 500 ms
   "2080TN450A01I02.FP_PARAM.AlarmDelay_L2_Acc" : Int AT %DB5124.DBW130, 500 ms
   "2080TN450A01I02.FP_PARAM.AlarmDelay_L3_Pre" : Int AT %DB5124.DBW132, 500 ms
   "2080TN450A01I02.FP_PARAM.AlarmDelay_L3_Acc" : Int AT %DB5124.DBW134, 500 ms
   "2080TN450A01I02.FP_PARAM.OpenLoopDelay_Pre" : Int AT %DB5124.DBW136, 500 ms
   "2080TN450A01I02.FP_PARAM.OpenLoopDelay_Acc" : Int AT %DB5124.DBW138, 500 ms
   "2080TN450A01I02.FP_PARAM.OverRangeDelay_Pre" : Int AT %DB5124.DBW140, 500 ms
   "2080TN450A01I02.FP_PARAM.OverRangeDelay_Acc" : Int AT %DB5124.DBW142, 500 ms
   "2080TN450A01I02.FP_PARAM.AuxLimit_H2_Value" : Real AT %DB5124.DBD144, 500 ms
   "2080TN450A01I02.FP_PARAM.AuxLimit_H1_Value" : Real AT %DB5124.DBD148, 500 ms
   "2080TN450A01I02.FP_PARAM.AuxLimit_L2_Value" : Real AT %DB5124.DBD152, 500 ms
   "2080TN450A01I02.FP_PARAM.AuxLimit_L1_Value" : Real AT %DB5124.DBD156, 500 ms
   "2080TN450A01I02.Unit" : TextRef, internal   // Еденицы измерения При експорте из ECS через скрипт заполняется автоматически, если теги копируются в ручную то требуется задатать свойство Text
   "2080TN450A01I02.Decimals" : TextRef, internal   // Формат отображения При експорте из ECS через скрипт, заполняется автоматически. Если теги копируются в ручную то требуется задатать свойство Text s999999.9
   "2080TN450A01I02.FP_EN.Square" : Bool AT %DB5124.DBX46.0, 500 ms
   "2080TN450A01I02.FP_EN.SquareRoot" : Bool AT %DB5124.DBX46.1, 500 ms
   "2080TN450A01I02.FP_EN.ParentSupress" : Bool AT %DB5124.DBX46.2, 500 ms
   "2080TN450A01I02.FP_EN.ParentSupressUnit" : Bool AT %DB5124.DBX46.3, 500 ms
   "2080TN450A01I02.FP_EN.Force" : Bool AT %DB5124.DBX46.4, 500 ms
   "2080TN450A01I02.FP_EN.Damping" : Bool AT %DB5124.DBX46.5, 500 ms
   "2080TN450A01I02.FP_EN.Gradient_Pos" : Bool AT %DB5124.DBX46.6, 500 ms
   "2080TN450A01I02.FP_EN.Gradient_Neg" : Bool AT %DB5124.DBX46.7, 500 ms
   "2080TN450A01I02.FP_EN.Hysteresis" : Bool AT %DB5124.DBX47.0, 500 ms
   "2080TN450A01I02.FP_EN.Alarm_H3" : Bool AT %DB5124.DBX47.1, 500 ms
   "2080TN450A01I02.FP_EN.Alarm_H2" : Bool AT %DB5124.DBX47.2, 500 ms
   "2080TN450A01I02.FP_EN.Alarm_H1" : Bool AT %DB5124.DBX47.3, 500 ms
   "2080TN450A01I02.FP_EN.Alarm_L1" : Bool AT %DB5124.DBX47.4, 500 ms
   "2080TN450A01I02.FP_EN.Alarm_L2" : Bool AT %DB5124.DBX47.5, 500 ms
   "2080TN450A01I02.FP_EN.Alarm_L3" : Bool AT %DB5124.DBX47.6, 500 ms
   "2080TN450A01I02.FP_EN.AlarmDelay_H3" : Bool AT %DB5124.DBX47.7, 500 ms
   "2080TN450A01I02.FP_EN.AlarmDelay_H2" : Bool AT %DB5124.DBX48.0, 500 ms
   "2080TN450A01I02.FP_EN.AlarmDelay_H1" : Bool AT %DB5124.DBX48.1, 500 ms
   "2080TN450A01I02.FP_EN.AlarmDelay_L1" : Bool AT %DB5124.DBX48.2, 500 ms
   "2080TN450A01I02.FP_EN.AlarmDelay_L2" : Bool AT %DB5124.DBX48.3, 500 ms
   "2080TN450A01I02.FP_EN.AlarmDelay_L3" : Bool AT %DB5124.DBX48.4, 500 ms
   "2080TN450A01I02.FP_EN.ROC_Warn" : Bool AT %DB5124.DBX48.5, 500 ms
   "2080TN450A01I02.FP_EN.U_Range_Warn" : Bool AT %DB5124.DBX48.6, 500 ms
   "2080TN450A01I02.FP_EN.O_Range_Warn" : Bool AT %DB5124.DBX48.7, 500 ms
   "2080TN450A01I02.trend_tag_name" : TextRef, internal   // Еденицы измерения При експорте из ECS через скрипт - заполняется автоматически, если теги копируются в ручную то требуется задатать свойство Text - имя тега для тренда
   "2080TN450A01I02.DQ.AL_H3" : Bool AT %DB5124.DBX16.0, 500 ms
   "2080TN450A01I02.DQ.AL_H2" : Bool AT %DB5124.DBX16.1, 500 ms
   "2080TN450A01I02.DQ.AL_H1" : Bool AT %DB5124.DBX16.2, 500 ms
   "2080TN450A01I02.DQ.AL_L1" : Bool AT %DB5124.DBX16.3, 500 ms
   "2080TN450A01I02.DQ.AL_L2" : Bool AT %DB5124.DBX16.4, 500 ms
   "2080TN450A01I02.DQ.AL_L3" : Bool AT %DB5124.DBX16.5, 500 ms
   "2080TN450A01I02.DQ.SIG_OK" : Bool AT %DB5124.DBX16.6, 500 ms
   "2080TN450A01I02.DQ.LIM_H2" : Bool AT %DB5124.DBX16.7, 500 ms
   "2080TN450A01I02.DQ.LIM_H1" : Bool AT %DB5124.DBX17.0, 500 ms
   "2080TN450A01I02.DQ.LIM_L1" : Bool AT %DB5124.DBX17.1, 500 ms
   "2080TN450A01I02.DQ.LIM_L2" : Bool AT %DB5124.DBX17.2, 500 ms
   "2080TN450A01I02.DQ.GR_P" : Bool AT %DB5124.DBX17.3, 500 ms
   "2080TN450A01I02.DQ.GR_N" : Bool AT %DB5124.DBX17.4, 500 ms
   "2080TN450A01I02.I.IN" : Real AT %DB5124.DBD2, 500 ms
   "2080TN450A01I02.I.SIG_TYPE" : Int AT %DB5124.DBW0, 500 ms
   "2080TN450A01I02.I.FI_BUS" : Byte AT %DB5124.DBB6, 500 ms
   "2080TN450A01I02.DI.U_RANGE" : Bool AT %DB5124.DBX7.0, 500 ms
   "2080TN450A01I02.DI.O_RANGE" : Bool AT %DB5124.DBX7.1, 500 ms
   "2080TN450A01I02.DI.SIG_FAULT" : Bool AT %DB5124.DBX7.2, 500 ms
   "2080TN450A01I02.DI.EnConfig" : Bool AT %DB5124.DBX7.3, 500 ms
   "2080TN450A01I02.DI.AEN" : Bool AT %DB5124.DBX7.4, 500 ms
   "2080TN450A01I02.DI.AL_SUPR" : Bool AT %DB5124.DBX7.5, 500 ms
   "2080TN450A01I02.Q.PV_NORM" : Real AT %DB5124.DBD8, 500 ms
   "2080TN450A01I02.Q.PV_SCAL" : Real AT %DB5124.DBD12, 500 ms
   "2080TN450A01I02.ParentInfo" : TextRef, internal   // Имя родителя для попап окна, вкладка инфо. При експорте из ECS через скрипт заполняется автоматически, если теги копируются в ручную то требуется в ручную задатать свойство Start Value

HMI tags "2080TN450A01I03"
   "2080TN450A01I03.MSW" : 52809b66-421d-457f-8884-6f7a49d4e247 AT %DB5125.DBX18.0, 500 ms
   "2080TN450A01I03.DefaultText" : TextRef, internal   // Заголовок POPUP окна. При експорте из ECS через скрипт заполняется автоматически, если теги копируются в ручную то требуется в ручную задатать свойство Start Value
   "2080TN450A01I03.BlockInfo" : Array [0..2] of Int AT %DB5125.DBX38.0, 500 ms
   "2080TN450A01I03.StatusWork" : Int AT %DB5125.DBW242, 500 ms
   "2080TN450A01I03.FP_PARAM.DampingTime" : Int AT %DB5125.DBW50, 500 ms
   "2080TN450A01I03.FP_PARAM.Force_Value" : Real AT %DB5125.DBD52, 500 ms
   "2080TN450A01I03.FP_PARAM.Scale_Min" : Real AT %DB5125.DBD56, 500 ms
   "2080TN450A01I03.FP_PARAM.Scale_Max" : Real AT %DB5125.DBD60, 500 ms
   "2080TN450A01I03.FP_PARAM.Gradient" : Real AT %DB5125.DBD64, 500 ms
   "2080TN450A01I03.FP_PARAM.Grad_Pos" : Real AT %DB5125.DBD68, 500 ms
   "2080TN450A01I03.FP_PARAM.Grad_Neg" : Real AT %DB5125.DBD72, 500 ms
   "2080TN450A01I03.FP_PARAM.Grad_X" : Real AT %DB5125.DBD76, 500 ms
   "2080TN450A01I03.FP_PARAM.Gradient_Time_Pre" : Int AT %DB5125.DBW80, 500 ms
   "2080TN450A01I03.FP_PARAM.Gradient_Time_ACC" : Int AT %DB5125.DBW82, 500 ms
   "2080TN450A01I03.FP_PARAM.Alarm_Hyst" : Real AT %DB5125.DBD84, 500 ms
   "2080TN450A01I03.FP_PARAM.AlarmLimit_H3" : Real AT %DB5125.DBD88, 500 ms
   "2080TN450A01I03.FP_PARAM.AlarmLimit_H2" : Real AT %DB5125.DBD92, 500 ms
   "2080TN450A01I03.FP_PARAM.AlarmLimit_H1" : Real AT %DB5125.DBD96, 500 ms
   "2080TN450A01I03.FP_PARAM.AlarmLimit_L1" : Real AT %DB5125.DBD100, 500 ms
   "2080TN450A01I03.FP_PARAM.AlarmLimit_L2" : Real AT %DB5125.DBD104, 500 ms
   "2080TN450A01I03.FP_PARAM.AlarmLimit_L3" : Real AT %DB5125.DBD108, 500 ms
   "2080TN450A01I03.FP_PARAM.AlarmDelay_H3_Pre" : Int AT %DB5125.DBW112, 500 ms
   "2080TN450A01I03.FP_PARAM.AlarmDelay_H3_Acc" : Int AT %DB5125.DBW114, 500 ms
   "2080TN450A01I03.FP_PARAM.AlarmDelay_H2_Pre" : Int AT %DB5125.DBW116, 500 ms
   "2080TN450A01I03.FP_PARAM.AlarmDelay_H2_Acc" : Int AT %DB5125.DBW118, 500 ms
   "2080TN450A01I03.FP_PARAM.AlarmDelay_H1_Pre" : Int AT %DB5125.DBW120, 500 ms
   "2080TN450A01I03.FP_PARAM.AlarmDelay_H1_Acc" : Int AT %DB5125.DBW122, 500 ms
   "2080TN450A01I03.FP_PARAM.AlarmDelay_L1_Pre" : Int AT %DB5125.DBW124, 500 ms
   "2080TN450A01I03.FP_PARAM.AlarmDelay_L1_Acc" : Int AT %DB5125.DBW126, 500 ms
   "2080TN450A01I03.FP_PARAM.AlarmDelay_L2_Pre" : Int AT %DB5125.DBW128, 500 ms
   "2080TN450A01I03.FP_PARAM.AlarmDelay_L2_Acc" : Int AT %DB5125.DBW130, 500 ms
   "2080TN450A01I03.FP_PARAM.AlarmDelay_L3_Pre" : Int AT %DB5125.DBW132, 500 ms
   "2080TN450A01I03.FP_PARAM.AlarmDelay_L3_Acc" : Int AT %DB5125.DBW134, 500 ms
   "2080TN450A01I03.FP_PARAM.OpenLoopDelay_Pre" : Int AT %DB5125.DBW136, 500 ms
   "2080TN450A01I03.FP_PARAM.OpenLoopDelay_Acc" : Int AT %DB5125.DBW138, 500 ms
   "2080TN450A01I03.FP_PARAM.OverRangeDelay_Pre" : Int AT %DB5125.DBW140, 500 ms
   "2080TN450A01I03.FP_PARAM.OverRangeDelay_Acc" : Int AT %DB5125.DBW142, 500 ms
   "2080TN450A01I03.FP_PARAM.AuxLimit_H2_Value" : Real AT %DB5125.DBD144, 500 ms
   "2080TN450A01I03.FP_PARAM.AuxLimit_H1_Value" : Real AT %DB5125.DBD148, 500 ms
   "2080TN450A01I03.FP_PARAM.AuxLimit_L2_Value" : Real AT %DB5125.DBD152, 500 ms
   "2080TN450A01I03.FP_PARAM.AuxLimit_L1_Value" : Real AT %DB5125.DBD156, 500 ms
   "2080TN450A01I03.Unit" : TextRef, internal   // Еденицы измерения При експорте из ECS через скрипт заполняется автоматически, если теги копируются в ручную то требуется задатать свойство Text
   "2080TN450A01I03.Decimals" : TextRef, internal   // Формат отображения При експорте из ECS через скрипт, заполняется автоматически. Если теги копируются в ручную то требуется задатать свойство Text s999999.9
   "2080TN450A01I03.FP_EN.Square" : Bool AT %DB5125.DBX46.0, 500 ms
   "2080TN450A01I03.FP_EN.SquareRoot" : Bool AT %DB5125.DBX46.1, 500 ms
   "2080TN450A01I03.FP_EN.ParentSupress" : Bool AT %DB5125.DBX46.2, 500 ms
   "2080TN450A01I03.FP_EN.ParentSupressUnit" : Bool AT %DB5125.DBX46.3, 500 ms
   "2080TN450A01I03.FP_EN.Force" : Bool AT %DB5125.DBX46.4, 500 ms
   "2080TN450A01I03.FP_EN.Damping" : Bool AT %DB5125.DBX46.5, 500 ms
   "2080TN450A01I03.FP_EN.Gradient_Pos" : Bool AT %DB5125.DBX46.6, 500 ms
   "2080TN450A01I03.FP_EN.Gradient_Neg" : Bool AT %DB5125.DBX46.7, 500 ms
   "2080TN450A01I03.FP_EN.Hysteresis" : Bool AT %DB5125.DBX47.0, 500 ms
   "2080TN450A01I03.FP_EN.Alarm_H3" : Bool AT %DB5125.DBX47.1, 500 ms
   "2080TN450A01I03.FP_EN.Alarm_H2" : Bool AT %DB5125.DBX47.2, 500 ms
   "2080TN450A01I03.FP_EN.Alarm_H1" : Bool AT %DB5125.DBX47.3, 500 ms
   "2080TN450A01I03.FP_EN.Alarm_L1" : Bool AT %DB5125.DBX47.4, 500 ms
   "2080TN450A01I03.FP_EN.Alarm_L2" : Bool AT %DB5125.DBX47.5, 500 ms
   "2080TN450A01I03.FP_EN.Alarm_L3" : Bool AT %DB5125.DBX47.6, 500 ms
   "2080TN450A01I03.FP_EN.AlarmDelay_H3" : Bool AT %DB5125.DBX47.7, 500 ms
   "2080TN450A01I03.FP_EN.AlarmDelay_H2" : Bool AT %DB5125.DBX48.0, 500 ms
   "2080TN450A01I03.FP_EN.AlarmDelay_H1" : Bool AT %DB5125.DBX48.1, 500 ms
   "2080TN450A01I03.FP_EN.AlarmDelay_L1" : Bool AT %DB5125.DBX48.2, 500 ms
   "2080TN450A01I03.FP_EN.AlarmDelay_L2" : Bool AT %DB5125.DBX48.3, 500 ms
   "2080TN450A01I03.FP_EN.AlarmDelay_L3" : Bool AT %DB5125.DBX48.4, 500 ms
   "2080TN450A01I03.FP_EN.ROC_Warn" : Bool AT %DB5125.DBX48.5, 500 ms
   "2080TN450A01I03.FP_EN.U_Range_Warn" : Bool AT %DB5125.DBX48.6, 500 ms
   "2080TN450A01I03.FP_EN.O_Range_Warn" : Bool AT %DB5125.DBX48.7, 500 ms
   "2080TN450A01I03.trend_tag_name" : TextRef, internal   // Еденицы измерения При експорте из ECS через скрипт - заполняется автоматически, если теги копируются в ручную то требуется задатать свойство Text - имя тега для тренда
   "2080TN450A01I03.DQ.AL_H3" : Bool AT %DB5125.DBX16.0, 500 ms
   "2080TN450A01I03.DQ.AL_H2" : Bool AT %DB5125.DBX16.1, 500 ms
   "2080TN450A01I03.DQ.AL_H1" : Bool AT %DB5125.DBX16.2, 500 ms
   "2080TN450A01I03.DQ.AL_L1" : Bool AT %DB5125.DBX16.3, 500 ms
   "2080TN450A01I03.DQ.AL_L2" : Bool AT %DB5125.DBX16.4, 500 ms
   "2080TN450A01I03.DQ.AL_L3" : Bool AT %DB5125.DBX16.5, 500 ms
   "2080TN450A01I03.DQ.SIG_OK" : Bool AT %DB5125.DBX16.6, 500 ms
   "2080TN450A01I03.DQ.LIM_H2" : Bool AT %DB5125.DBX16.7, 500 ms
   "2080TN450A01I03.DQ.LIM_H1" : Bool AT %DB5125.DBX17.0, 500 ms
   "2080TN450A01I03.DQ.LIM_L1" : Bool AT %DB5125.DBX17.1, 500 ms
   "2080TN450A01I03.DQ.LIM_L2" : Bool AT %DB5125.DBX17.2, 500 ms
   "2080TN450A01I03.DQ.GR_P" : Bool AT %DB5125.DBX17.3, 500 ms
   "2080TN450A01I03.DQ.GR_N" : Bool AT %DB5125.DBX17.4, 500 ms
   "2080TN450A01I03.I.IN" : Real AT %DB5125.DBD2, 500 ms
   "2080TN450A01I03.I.SIG_TYPE" : Int AT %DB5125.DBW0, 500 ms
   "2080TN450A01I03.I.FI_BUS" : Byte AT %DB5125.DBB6, 500 ms
   "2080TN450A01I03.DI.U_RANGE" : Bool AT %DB5125.DBX7.0, 500 ms
   "2080TN450A01I03.DI.O_RANGE" : Bool AT %DB5125.DBX7.1, 500 ms
   "2080TN450A01I03.DI.SIG_FAULT" : Bool AT %DB5125.DBX7.2, 500 ms
   "2080TN450A01I03.DI.EnConfig" : Bool AT %DB5125.DBX7.3, 500 ms
   "2080TN450A01I03.DI.AEN" : Bool AT %DB5125.DBX7.4, 500 ms
   "2080TN450A01I03.DI.AL_SUPR" : Bool AT %DB5125.DBX7.5, 500 ms
   "2080TN450A01I03.Q.PV_NORM" : Real AT %DB5125.DBD8, 500 ms
   "2080TN450A01I03.Q.PV_SCAL" : Real AT %DB5125.DBD12, 500 ms
   "2080TN450A01I03.ParentInfo" : TextRef, internal   // Имя родителя для попап окна, вкладка инфо. При експорте из ECS через скрипт заполняется автоматически, если теги копируются в ручную то требуется в ручную задатать свойство Start Value

HMI tags "2080TN450A01I04"
   "2080TN450A01I04.MSW" : 52809b66-421d-457f-8884-6f7a49d4e247 AT %DB5126.DBX18.0, 500 ms
   "2080TN450A01I04.DefaultText" : TextRef, internal   // Заголовок POPUP окна. При експорте из ECS через скрипт заполняется автоматически, если теги копируются в ручную то требуется в ручную задатать свойство Start Value
   "2080TN450A01I04.BlockInfo" : Array [0..2] of Int AT %DB5126.DBX38.0, 500 ms
   "2080TN450A01I04.StatusWork" : Int AT %DB5126.DBW242, 500 ms
   "2080TN450A01I04.FP_PARAM.DampingTime" : Int AT %DB5126.DBW50, 500 ms
   "2080TN450A01I04.FP_PARAM.Force_Value" : Real AT %DB5126.DBD52, 500 ms
   "2080TN450A01I04.FP_PARAM.Scale_Min" : Real AT %DB5126.DBD56, 500 ms
   "2080TN450A01I04.FP_PARAM.Scale_Max" : Real AT %DB5126.DBD60, 500 ms
   "2080TN450A01I04.FP_PARAM.Gradient" : Real AT %DB5126.DBD64, 500 ms
   "2080TN450A01I04.FP_PARAM.Grad_Pos" : Real AT %DB5126.DBD68, 500 ms
   "2080TN450A01I04.FP_PARAM.Grad_Neg" : Real AT %DB5126.DBD72, 500 ms
   "2080TN450A01I04.FP_PARAM.Grad_X" : Real AT %DB5126.DBD76, 500 ms
   "2080TN450A01I04.FP_PARAM.Gradient_Time_Pre" : Int AT %DB5126.DBW80, 500 ms
   "2080TN450A01I04.FP_PARAM.Gradient_Time_ACC" : Int AT %DB5126.DBW82, 500 ms
   "2080TN450A01I04.FP_PARAM.Alarm_Hyst" : Real AT %DB5126.DBD84, 500 ms
   "2080TN450A01I04.FP_PARAM.AlarmLimit_H3" : Real AT %DB5126.DBD88, 500 ms
   "2080TN450A01I04.FP_PARAM.AlarmLimit_H2" : Real AT %DB5126.DBD92, 500 ms
   "2080TN450A01I04.FP_PARAM.AlarmLimit_H1" : Real AT %DB5126.DBD96, 500 ms
   "2080TN450A01I04.FP_PARAM.AlarmLimit_L1" : Real AT %DB5126.DBD100, 500 ms
   "2080TN450A01I04.FP_PARAM.AlarmLimit_L2" : Real AT %DB5126.DBD104, 500 ms
   "2080TN450A01I04.FP_PARAM.AlarmLimit_L3" : Real AT %DB5126.DBD108, 500 ms
   "2080TN450A01I04.FP_PARAM.AlarmDelay_H3_Pre" : Int AT %DB5126.DBW112, 500 ms
   "2080TN450A01I04.FP_PARAM.AlarmDelay_H3_Acc" : Int AT %DB5126.DBW114, 500 ms
   "2080TN450A01I04.FP_PARAM.AlarmDelay_H2_Pre" : Int AT %DB5126.DBW116, 500 ms
   "2080TN450A01I04.FP_PARAM.AlarmDelay_H2_Acc" : Int AT %DB5126.DBW118, 500 ms
   "2080TN450A01I04.FP_PARAM.AlarmDelay_H1_Pre" : Int AT %DB5126.DBW120, 500 ms
   "2080TN450A01I04.FP_PARAM.AlarmDelay_H1_Acc" : Int AT %DB5126.DBW122, 500 ms
   "2080TN450A01I04.FP_PARAM.AlarmDelay_L1_Pre" : Int AT %DB5126.DBW124, 500 ms
   "2080TN450A01I04.FP_PARAM.AlarmDelay_L1_Acc" : Int AT %DB5126.DBW126, 500 ms
   "2080TN450A01I04.FP_PARAM.AlarmDelay_L2_Pre" : Int AT %DB5126.DBW128, 500 ms
   "2080TN450A01I04.FP_PARAM.AlarmDelay_L2_Acc" : Int AT %DB5126.DBW130, 500 ms
   "2080TN450A01I04.FP_PARAM.AlarmDelay_L3_Pre" : Int AT %DB5126.DBW132, 500 ms
   "2080TN450A01I04.FP_PARAM.AlarmDelay_L3_Acc" : Int AT %DB5126.DBW134, 500 ms
   "2080TN450A01I04.FP_PARAM.OpenLoopDelay_Pre" : Int AT %DB5126.DBW136, 500 ms
   "2080TN450A01I04.FP_PARAM.OpenLoopDelay_Acc" : Int AT %DB5126.DBW138, 500 ms
   "2080TN450A01I04.FP_PARAM.OverRangeDelay_Pre" : Int AT %DB5126.DBW140, 500 ms
   "2080TN450A01I04.FP_PARAM.OverRangeDelay_Acc" : Int AT %DB5126.DBW142, 500 ms
   "2080TN450A01I04.FP_PARAM.AuxLimit_H2_Value" : Real AT %DB5126.DBD144, 500 ms
   "2080TN450A01I04.FP_PARAM.AuxLimit_H1_Value" : Real AT %DB5126.DBD148, 500 ms
   "2080TN450A01I04.FP_PARAM.AuxLimit_L2_Value" : Real AT %DB5126.DBD152, 500 ms
   "2080TN450A01I04.FP_PARAM.AuxLimit_L1_Value" : Real AT %DB5126.DBD156, 500 ms
   "2080TN450A01I04.Unit" : TextRef, internal   // Еденицы измерения При експорте из ECS через скрипт заполняется автоматически, если теги копируются в ручную то требуется задатать свойство Text
   "2080TN450A01I04.Decimals" : TextRef, internal   // Формат отображения При експорте из ECS через скрипт, заполняется автоматически. Если теги копируются в ручную то требуется задатать свойство Text s999999.9
   "2080TN450A01I04.FP_EN.Square" : Bool AT %DB5126.DBX46.0, 500 ms
   "2080TN450A01I04.FP_EN.SquareRoot" : Bool AT %DB5126.DBX46.1, 500 ms
   "2080TN450A01I04.FP_EN.ParentSupress" : Bool AT %DB5126.DBX46.2, 500 ms
   "2080TN450A01I04.FP_EN.ParentSupressUnit" : Bool AT %DB5126.DBX46.3, 500 ms
   "2080TN450A01I04.FP_EN.Force" : Bool AT %DB5126.DBX46.4, 500 ms
   "2080TN450A01I04.FP_EN.Damping" : Bool AT %DB5126.DBX46.5, 500 ms
   "2080TN450A01I04.FP_EN.Gradient_Pos" : Bool AT %DB5126.DBX46.6, 500 ms
   "2080TN450A01I04.FP_EN.Gradient_Neg" : Bool AT %DB5126.DBX46.7, 500 ms
   "2080TN450A01I04.FP_EN.Hysteresis" : Bool AT %DB5126.DBX47.0, 500 ms
   "2080TN450A01I04.FP_EN.Alarm_H3" : Bool AT %DB5126.DBX47.1, 500 ms
   "2080TN450A01I04.FP_EN.Alarm_H2" : Bool AT %DB5126.DBX47.2, 500 ms
   "2080TN450A01I04.FP_EN.Alarm_H1" : Bool AT %DB5126.DBX47.3, 500 ms
   "2080TN450A01I04.FP_EN.Alarm_L1" : Bool AT %DB5126.DBX47.4, 500 ms
   "2080TN450A01I04.FP_EN.Alarm_L2" : Bool AT %DB5126.DBX47.5, 500 ms
   "2080TN450A01I04.FP_EN.Alarm_L3" : Bool AT %DB5126.DBX47.6, 500 ms
   "2080TN450A01I04.FP_EN.AlarmDelay_H3" : Bool AT %DB5126.DBX47.7, 500 ms
   "2080TN450A01I04.FP_EN.AlarmDelay_H2" : Bool AT %DB5126.DBX48.0, 500 ms
   "2080TN450A01I04.FP_EN.AlarmDelay_H1" : Bool AT %DB5126.DBX48.1, 500 ms
   "2080TN450A01I04.FP_EN.AlarmDelay_L1" : Bool AT %DB5126.DBX48.2, 500 ms
   "2080TN450A01I04.FP_EN.AlarmDelay_L2" : Bool AT %DB5126.DBX48.3, 500 ms
   "2080TN450A01I04.FP_EN.AlarmDelay_L3" : Bool AT %DB5126.DBX48.4, 500 ms
   "2080TN450A01I04.FP_EN.ROC_Warn" : Bool AT %DB5126.DBX48.5, 500 ms
   "2080TN450A01I04.FP_EN.U_Range_Warn" : Bool AT %DB5126.DBX48.6, 500 ms
   "2080TN450A01I04.FP_EN.O_Range_Warn" : Bool AT %DB5126.DBX48.7, 500 ms
   "2080TN450A01I04.trend_tag_name" : TextRef, internal   // Еденицы измерения При експорте из ECS через скрипт - заполняется автоматически, если теги копируются в ручную то требуется задатать свойство Text - имя тега для тренда
   "2080TN450A01I04.DQ.AL_H3" : Bool AT %DB5126.DBX16.0, 500 ms
   "2080TN450A01I04.DQ.AL_H2" : Bool AT %DB5126.DBX16.1, 500 ms
   "2080TN450A01I04.DQ.AL_H1" : Bool AT %DB5126.DBX16.2, 500 ms
   "2080TN450A01I04.DQ.AL_L1" : Bool AT %DB5126.DBX16.3, 500 ms
   "2080TN450A01I04.DQ.AL_L2" : Bool AT %DB5126.DBX16.4, 500 ms
   "2080TN450A01I04.DQ.AL_L3" : Bool AT %DB5126.DBX16.5, 500 ms
   "2080TN450A01I04.DQ.SIG_OK" : Bool AT %DB5126.DBX16.6, 500 ms
   "2080TN450A01I04.DQ.LIM_H2" : Bool AT %DB5126.DBX16.7, 500 ms
   "2080TN450A01I04.DQ.LIM_H1" : Bool AT %DB5126.DBX17.0, 500 ms
   "2080TN450A01I04.DQ.LIM_L1" : Bool AT %DB5126.DBX17.1, 500 ms
   "2080TN450A01I04.DQ.LIM_L2" : Bool AT %DB5126.DBX17.2, 500 ms
   "2080TN450A01I04.DQ.GR_P" : Bool AT %DB5126.DBX17.3, 500 ms
   "2080TN450A01I04.DQ.GR_N" : Bool AT %DB5126.DBX17.4, 500 ms
   "2080TN450A01I04.I.IN" : Real AT %DB5126.DBD2, 500 ms
   "2080TN450A01I04.I.SIG_TYPE" : Int AT %DB5126.DBW0, 500 ms
   "2080TN450A01I04.I.FI_BUS" : Byte AT %DB5126.DBB6, 500 ms
   "2080TN450A01I04.DI.U_RANGE" : Bool AT %DB5126.DBX7.0, 500 ms
   "2080TN450A01I04.DI.O_RANGE" : Bool AT %DB5126.DBX7.1, 500 ms
   "2080TN450A01I04.DI.SIG_FAULT" : Bool AT %DB5126.DBX7.2, 500 ms
   "2080TN450A01I04.DI.EnConfig" : Bool AT %DB5126.DBX7.3, 500 ms
   "2080TN450A01I04.DI.AEN" : Bool AT %DB5126.DBX7.4, 500 ms
   "2080TN450A01I04.DI.AL_SUPR" : Bool AT %DB5126.DBX7.5, 500 ms
   "2080TN450A01I04.Q.PV_NORM" : Real AT %DB5126.DBD8, 500 ms
   "2080TN450A01I04.Q.PV_SCAL" : Real AT %DB5126.DBD12, 500 ms
   "2080TN450A01I04.ParentInfo" : TextRef, internal   // Имя родителя для попап окна, вкладка инфо. При експорте из ECS через скрипт заполняется автоматически, если теги копируются в ручную то требуется в ручную задатать свойство Start Value

HMI tags "2080TN450A01L01"
   "2080TN450A01L01.MSW" : 52809b66-421d-457f-8884-6f7a49d4e247 AT %DB5127.DBX18.0, 500 ms
   "2080TN450A01L01.DefaultText" : TextRef, internal   // Заголовок POPUP окна. При експорте из ECS через скрипт заполняется автоматически, если теги копируются в ручную то требуется в ручную задатать свойство Start Value
   "2080TN450A01L01.BlockInfo" : Array [0..2] of Int AT %DB5127.DBX38.0, 500 ms
   "2080TN450A01L01.StatusWork" : Int AT %DB5127.DBW242, 500 ms
   "2080TN450A01L01.FP_PARAM.DampingTime" : Int AT %DB5127.DBW50, 500 ms
   "2080TN450A01L01.FP_PARAM.Force_Value" : Real AT %DB5127.DBD52, 500 ms
   "2080TN450A01L01.FP_PARAM.Scale_Min" : Real AT %DB5127.DBD56, 500 ms
   "2080TN450A01L01.FP_PARAM.Scale_Max" : Real AT %DB5127.DBD60, 500 ms
   "2080TN450A01L01.FP_PARAM.Gradient" : Real AT %DB5127.DBD64, 500 ms
   "2080TN450A01L01.FP_PARAM.Grad_Pos" : Real AT %DB5127.DBD68, 500 ms
   "2080TN450A01L01.FP_PARAM.Grad_Neg" : Real AT %DB5127.DBD72, 500 ms
   "2080TN450A01L01.FP_PARAM.Grad_X" : Real AT %DB5127.DBD76, 500 ms
   "2080TN450A01L01.FP_PARAM.Gradient_Time_Pre" : Int AT %DB5127.DBW80, 500 ms
   "2080TN450A01L01.FP_PARAM.Gradient_Time_ACC" : Int AT %DB5127.DBW82, 500 ms
   "2080TN450A01L01.FP_PARAM.Alarm_Hyst" : Real AT %DB5127.DBD84, 500 ms
   "2080TN450A01L01.FP_PARAM.AlarmLimit_H3" : Real AT %DB5127.DBD88, 500 ms
   "2080TN450A01L01.FP_PARAM.AlarmLimit_H2" : Real AT %DB5127.DBD92, 500 ms
   "2080TN450A01L01.FP_PARAM.AlarmLimit_H1" : Real AT %DB5127.DBD96, 500 ms
   "2080TN450A01L01.FP_PARAM.AlarmLimit_L1" : Real AT %DB5127.DBD100, 500 ms
   "2080TN450A01L01.FP_PARAM.AlarmLimit_L2" : Real AT %DB5127.DBD104, 500 ms
   "2080TN450A01L01.FP_PARAM.AlarmLimit_L3" : Real AT %DB5127.DBD108, 500 ms
   "2080TN450A01L01.FP_PARAM.AlarmDelay_H3_Pre" : Int AT %DB5127.DBW112, 500 ms
   "2080TN450A01L01.FP_PARAM.AlarmDelay_H3_Acc" : Int AT %DB5127.DBW114, 500 ms
   "2080TN450A01L01.FP_PARAM.AlarmDelay_H2_Pre" : Int AT %DB5127.DBW116, 500 ms
   "2080TN450A01L01.FP_PARAM.AlarmDelay_H2_Acc" : Int AT %DB5127.DBW118, 500 ms
   "2080TN450A01L01.FP_PARAM.AlarmDelay_H1_Pre" : Int AT %DB5127.DBW120, 500 ms
   "2080TN450A01L01.FP_PARAM.AlarmDelay_H1_Acc" : Int AT %DB5127.DBW122, 500 ms
   "2080TN450A01L01.FP_PARAM.AlarmDelay_L1_Pre" : Int AT %DB5127.DBW124, 500 ms
   "2080TN450A01L01.FP_PARAM.AlarmDelay_L1_Acc" : Int AT %DB5127.DBW126, 500 ms
   "2080TN450A01L01.FP_PARAM.AlarmDelay_L2_Pre" : Int AT %DB5127.DBW128, 500 ms
   "2080TN450A01L01.FP_PARAM.AlarmDelay_L2_Acc" : Int AT %DB5127.DBW130, 500 ms
   "2080TN450A01L01.FP_PARAM.AlarmDelay_L3_Pre" : Int AT %DB5127.DBW132, 500 ms
   "2080TN450A01L01.FP_PARAM.AlarmDelay_L3_Acc" : Int AT %DB5127.DBW134, 500 ms
   "2080TN450A01L01.FP_PARAM.OpenLoopDelay_Pre" : Int AT %DB5127.DBW136, 500 ms
   "2080TN450A01L01.FP_PARAM.OpenLoopDelay_Acc" : Int AT %DB5127.DBW138, 500 ms
   "2080TN450A01L01.FP_PARAM.OverRangeDelay_Pre" : Int AT %DB5127.DBW140, 500 ms
   "2080TN450A01L01.FP_PARAM.OverRangeDelay_Acc" : Int AT %DB5127.DBW142, 500 ms
   "2080TN450A01L01.FP_PARAM.AuxLimit_H2_Value" : Real AT %DB5127.DBD144, 500 ms
   "2080TN450A01L01.FP_PARAM.AuxLimit_H1_Value" : Real AT %DB5127.DBD148, 500 ms
   "2080TN450A01L01.FP_PARAM.AuxLimit_L2_Value" : Real AT %DB5127.DBD152, 500 ms
   "2080TN450A01L01.FP_PARAM.AuxLimit_L1_Value" : Real AT %DB5127.DBD156, 500 ms
   "2080TN450A01L01.Unit" : TextRef, internal   // Еденицы измерения При експорте из ECS через скрипт заполняется автоматически, если теги копируются в ручную то требуется задатать свойство Text
   "2080TN450A01L01.Decimals" : TextRef, internal   // Формат отображения При експорте из ECS через скрипт, заполняется автоматически. Если теги копируются в ручную то требуется задатать свойство Text s999999.9
   "2080TN450A01L01.FP_EN.Square" : Bool AT %DB5127.DBX46.0, 500 ms
   "2080TN450A01L01.FP_EN.SquareRoot" : Bool AT %DB5127.DBX46.1, 500 ms
   "2080TN450A01L01.FP_EN.ParentSupress" : Bool AT %DB5127.DBX46.2, 500 ms
   "2080TN450A01L01.FP_EN.ParentSupressUnit" : Bool AT %DB5127.DBX46.3, 500 ms
   "2080TN450A01L01.FP_EN.Force" : Bool AT %DB5127.DBX46.4, 500 ms
   "2080TN450A01L01.FP_EN.Damping" : Bool AT %DB5127.DBX46.5, 500 ms
   "2080TN450A01L01.FP_EN.Gradient_Pos" : Bool AT %DB5127.DBX46.6, 500 ms
   "2080TN450A01L01.FP_EN.Gradient_Neg" : Bool AT %DB5127.DBX46.7, 500 ms
   "2080TN450A01L01.FP_EN.Hysteresis" : Bool AT %DB5127.DBX47.0, 500 ms
   "2080TN450A01L01.FP_EN.Alarm_H3" : Bool AT %DB5127.DBX47.1, 500 ms
   "2080TN450A01L01.FP_EN.Alarm_H2" : Bool AT %DB5127.DBX47.2, 500 ms
   "2080TN450A01L01.FP_EN.Alarm_H1" : Bool AT %DB5127.DBX47.3, 500 ms
   "2080TN450A01L01.FP_EN.Alarm_L1" : Bool AT %DB5127.DBX47.4, 500 ms
   "2080TN450A01L01.FP_EN.Alarm_L2" : Bool AT %DB5127.DBX47.5, 500 ms
   "2080TN450A01L01.FP_EN.Alarm_L3" : Bool AT %DB5127.DBX47.6, 500 ms
   "2080TN450A01L01.FP_EN.AlarmDelay_H3" : Bool AT %DB5127.DBX47.7, 500 ms
   "2080TN450A01L01.FP_EN.AlarmDelay_H2" : Bool AT %DB5127.DBX48.0, 500 ms
   "2080TN450A01L01.FP_EN.AlarmDelay_H1" : Bool AT %DB5127.DBX48.1, 500 ms
   "2080TN450A01L01.FP_EN.AlarmDelay_L1" : Bool AT %DB5127.DBX48.2, 500 ms
   "2080TN450A01L01.FP_EN.AlarmDelay_L2" : Bool AT %DB5127.DBX48.3, 500 ms
   "2080TN450A01L01.FP_EN.AlarmDelay_L3" : Bool AT %DB5127.DBX48.4, 500 ms
   "2080TN450A01L01.FP_EN.ROC_Warn" : Bool AT %DB5127.DBX48.5, 500 ms
   "2080TN450A01L01.FP_EN.U_Range_Warn" : Bool AT %DB5127.DBX48.6, 500 ms
   "2080TN450A01L01.FP_EN.O_Range_Warn" : Bool AT %DB5127.DBX48.7, 500 ms
   "2080TN450A01L01.trend_tag_name" : TextRef, internal   // Еденицы измерения При експорте из ECS через скрипт - заполняется автоматически, если теги копируются в ручную то требуется задатать свойство Text - имя тега для тренда
   "2080TN450A01L01.DQ.AL_H3" : Bool AT %DB5127.DBX16.0, 500 ms
   "2080TN450A01L01.DQ.AL_H2" : Bool AT %DB5127.DBX16.1, 500 ms
   "2080TN450A01L01.DQ.AL_H1" : Bool AT %DB5127.DBX16.2, 500 ms
   "2080TN450A01L01.DQ.AL_L1" : Bool AT %DB5127.DBX16.3, 500 ms
   "2080TN450A01L01.DQ.AL_L2" : Bool AT %DB5127.DBX16.4, 500 ms
   "2080TN450A01L01.DQ.AL_L3" : Bool AT %DB5127.DBX16.5, 500 ms
   "2080TN450A01L01.DQ.SIG_OK" : Bool AT %DB5127.DBX16.6, 500 ms
   "2080TN450A01L01.DQ.LIM_H2" : Bool AT %DB5127.DBX16.7, 500 ms
   "2080TN450A01L01.DQ.LIM_H1" : Bool AT %DB5127.DBX17.0, 500 ms
   "2080TN450A01L01.DQ.LIM_L1" : Bool AT %DB5127.DBX17.1, 500 ms
   "2080TN450A01L01.DQ.LIM_L2" : Bool AT %DB5127.DBX17.2, 500 ms
   "2080TN450A01L01.DQ.GR_P" : Bool AT %DB5127.DBX17.3, 500 ms
   "2080TN450A01L01.DQ.GR_N" : Bool AT %DB5127.DBX17.4, 500 ms
   "2080TN450A01L01.I.IN" : Real AT %DB5127.DBD2, 500 ms
   "2080TN450A01L01.I.SIG_TYPE" : Int AT %DB5127.DBW0, 500 ms
   "2080TN450A01L01.I.FI_BUS" : Byte AT %DB5127.DBB6, 500 ms
   "2080TN450A01L01.DI.U_RANGE" : Bool AT %DB5127.DBX7.0, 500 ms
   "2080TN450A01L01.DI.O_RANGE" : Bool AT %DB5127.DBX7.1, 500 ms
   "2080TN450A01L01.DI.SIG_FAULT" : Bool AT %DB5127.DBX7.2, 500 ms
   "2080TN450A01L01.DI.EnConfig" : Bool AT %DB5127.DBX7.3, 500 ms
   "2080TN450A01L01.DI.AEN" : Bool AT %DB5127.DBX7.4, 500 ms
   "2080TN450A01L01.DI.AL_SUPR" : Bool AT %DB5127.DBX7.5, 500 ms
   "2080TN450A01L01.Q.PV_NORM" : Real AT %DB5127.DBD8, 500 ms
   "2080TN450A01L01.Q.PV_SCAL" : Real AT %DB5127.DBD12, 500 ms
   "2080TN450A01L01.ParentInfo" : TextRef, internal   // Имя родителя для попап окна, вкладка инфо. При експорте из ECS через скрипт заполняется автоматически, если теги копируются в ручную то требуется в ручную задатать свойство Start Value

HMI tags "2080TN450A01Z01"
   "2080TN450A01Z01.MSW" : 52809b66-421d-457f-8884-6f7a49d4e247 AT %DB5128.DBX18.0, 500 ms
   "2080TN450A01Z01.DefaultText" : TextRef, internal   // Заголовок POPUP окна. При експорте из ECS через скрипт заполняется автоматически, если теги копируются в ручную то требуется в ручную задатать свойство Start Value
   "2080TN450A01Z01.BlockInfo" : Array [0..2] of Int AT %DB5128.DBX38.0, 500 ms
   "2080TN450A01Z01.StatusWork" : Int AT %DB5128.DBW242, 500 ms
   "2080TN450A01Z01.FP_PARAM.DampingTime" : Int AT %DB5128.DBW50, 500 ms
   "2080TN450A01Z01.FP_PARAM.Force_Value" : Real AT %DB5128.DBD52, 500 ms
   "2080TN450A01Z01.FP_PARAM.Scale_Min" : Real AT %DB5128.DBD56, 500 ms
   "2080TN450A01Z01.FP_PARAM.Scale_Max" : Real AT %DB5128.DBD60, 500 ms
   "2080TN450A01Z01.FP_PARAM.Gradient" : Real AT %DB5128.DBD64, 500 ms
   "2080TN450A01Z01.FP_PARAM.Grad_Pos" : Real AT %DB5128.DBD68, 500 ms
   "2080TN450A01Z01.FP_PARAM.Grad_Neg" : Real AT %DB5128.DBD72, 500 ms
   "2080TN450A01Z01.FP_PARAM.Grad_X" : Real AT %DB5128.DBD76, 500 ms
   "2080TN450A01Z01.FP_PARAM.Gradient_Time_Pre" : Int AT %DB5128.DBW80, 500 ms
   "2080TN450A01Z01.FP_PARAM.Gradient_Time_ACC" : Int AT %DB5128.DBW82, 500 ms
   "2080TN450A01Z01.FP_PARAM.Alarm_Hyst" : Real AT %DB5128.DBD84, 500 ms
   "2080TN450A01Z01.FP_PARAM.AlarmLimit_H3" : Real AT %DB5128.DBD88, 500 ms
   "2080TN450A01Z01.FP_PARAM.AlarmLimit_H2" : Real AT %DB5128.DBD92, 500 ms
   "2080TN450A01Z01.FP_PARAM.AlarmLimit_H1" : Real AT %DB5128.DBD96, 500 ms
   "2080TN450A01Z01.FP_PARAM.AlarmLimit_L1" : Real AT %DB5128.DBD100, 500 ms
   "2080TN450A01Z01.FP_PARAM.AlarmLimit_L2" : Real AT %DB5128.DBD104, 500 ms
   "2080TN450A01Z01.FP_PARAM.AlarmLimit_L3" : Real AT %DB5128.DBD108, 500 ms
   "2080TN450A01Z01.FP_PARAM.AlarmDelay_H3_Pre" : Int AT %DB5128.DBW112, 500 ms
   "2080TN450A01Z01.FP_PARAM.AlarmDelay_H3_Acc" : Int AT %DB5128.DBW114, 500 ms
   "2080TN450A01Z01.FP_PARAM.AlarmDelay_H2_Pre" : Int AT %DB5128.DBW116, 500 ms
   "2080TN450A01Z01.FP_PARAM.AlarmDelay_H2_Acc" : Int AT %DB5128.DBW118, 500 ms
   "2080TN450A01Z01.FP_PARAM.AlarmDelay_H1_Pre" : Int AT %DB5128.DBW120, 500 ms
   "2080TN450A01Z01.FP_PARAM.AlarmDelay_H1_Acc" : Int AT %DB5128.DBW122, 500 ms
   "2080TN450A01Z01.FP_PARAM.AlarmDelay_L1_Pre" : Int AT %DB5128.DBW124, 500 ms
   "2080TN450A01Z01.FP_PARAM.AlarmDelay_L1_Acc" : Int AT %DB5128.DBW126, 500 ms
   "2080TN450A01Z01.FP_PARAM.AlarmDelay_L2_Pre" : Int AT %DB5128.DBW128, 500 ms
   "2080TN450A01Z01.FP_PARAM.AlarmDelay_L2_Acc" : Int AT %DB5128.DBW130, 500 ms
   "2080TN450A01Z01.FP_PARAM.AlarmDelay_L3_Pre" : Int AT %DB5128.DBW132, 500 ms
   "2080TN450A01Z01.FP_PARAM.AlarmDelay_L3_Acc" : Int AT %DB5128.DBW134, 500 ms
   "2080TN450A01Z01.FP_PARAM.OpenLoopDelay_Pre" : Int AT %DB5128.DBW136, 500 ms
   "2080TN450A01Z01.FP_PARAM.OpenLoopDelay_Acc" : Int AT %DB5128.DBW138, 500 ms
   "2080TN450A01Z01.FP_PARAM.OverRangeDelay_Pre" : Int AT %DB5128.DBW140, 500 ms
   "2080TN450A01Z01.FP_PARAM.OverRangeDelay_Acc" : Int AT %DB5128.DBW142, 500 ms
   "2080TN450A01Z01.FP_PARAM.AuxLimit_H2_Value" : Real AT %DB5128.DBD144, 500 ms
   "2080TN450A01Z01.FP_PARAM.AuxLimit_H1_Value" : Real AT %DB5128.DBD148, 500 ms
   "2080TN450A01Z01.FP_PARAM.AuxLimit_L2_Value" : Real AT %DB5128.DBD152, 500 ms
   "2080TN450A01Z01.FP_PARAM.AuxLimit_L1_Value" : Real AT %DB5128.DBD156, 500 ms
   "2080TN450A01Z01.Unit" : TextRef, internal   // Еденицы измерения При експорте из ECS через скрипт заполняется автоматически, если теги копируются в ручную то требуется задатать свойство Text
   "2080TN450A01Z01.Decimals" : TextRef, internal   // Формат отображения При експорте из ECS через скрипт, заполняется автоматически. Если теги копируются в ручную то требуется задатать свойство Text s999999.9
   "2080TN450A01Z01.FP_EN.Square" : Bool AT %DB5128.DBX46.0, 500 ms
   "2080TN450A01Z01.FP_EN.SquareRoot" : Bool AT %DB5128.DBX46.1, 500 ms
   "2080TN450A01Z01.FP_EN.ParentSupress" : Bool AT %DB5128.DBX46.2, 500 ms
   "2080TN450A01Z01.FP_EN.ParentSupressUnit" : Bool AT %DB5128.DBX46.3, 500 ms
   "2080TN450A01Z01.FP_EN.Force" : Bool AT %DB5128.DBX46.4, 500 ms
   "2080TN450A01Z01.FP_EN.Damping" : Bool AT %DB5128.DBX46.5, 500 ms
   "2080TN450A01Z01.FP_EN.Gradient_Pos" : Bool AT %DB5128.DBX46.6, 500 ms
   "2080TN450A01Z01.FP_EN.Gradient_Neg" : Bool AT %DB5128.DBX46.7, 500 ms
   "2080TN450A01Z01.FP_EN.Hysteresis" : Bool AT %DB5128.DBX47.0, 500 ms
   "2080TN450A01Z01.FP_EN.Alarm_H3" : Bool AT %DB5128.DBX47.1, 500 ms
   "2080TN450A01Z01.FP_EN.Alarm_H2" : Bool AT %DB5128.DBX47.2, 500 ms
   "2080TN450A01Z01.FP_EN.Alarm_H1" : Bool AT %DB5128.DBX47.3, 500 ms
   "2080TN450A01Z01.FP_EN.Alarm_L1" : Bool AT %DB5128.DBX47.4, 500 ms
   "2080TN450A01Z01.FP_EN.Alarm_L2" : Bool AT %DB5128.DBX47.5, 500 ms
   "2080TN450A01Z01.FP_EN.Alarm_L3" : Bool AT %DB5128.DBX47.6, 500 ms
   "2080TN450A01Z01.FP_EN.AlarmDelay_H3" : Bool AT %DB5128.DBX47.7, 500 ms
   "2080TN450A01Z01.FP_EN.AlarmDelay_H2" : Bool AT %DB5128.DBX48.0, 500 ms
   "2080TN450A01Z01.FP_EN.AlarmDelay_H1" : Bool AT %DB5128.DBX48.1, 500 ms
   "2080TN450A01Z01.FP_EN.AlarmDelay_L1" : Bool AT %DB5128.DBX48.2, 500 ms
   "2080TN450A01Z01.FP_EN.AlarmDelay_L2" : Bool AT %DB5128.DBX48.3, 500 ms
   "2080TN450A01Z01.FP_EN.AlarmDelay_L3" : Bool AT %DB5128.DBX48.4, 500 ms
   "2080TN450A01Z01.FP_EN.ROC_Warn" : Bool AT %DB5128.DBX48.5, 500 ms
   "2080TN450A01Z01.FP_EN.U_Range_Warn" : Bool AT %DB5128.DBX48.6, 500 ms
   "2080TN450A01Z01.FP_EN.O_Range_Warn" : Bool AT %DB5128.DBX48.7, 500 ms
   "2080TN450A01Z01.trend_tag_name" : TextRef, internal   // Еденицы измерения При експорте из ECS через скрипт - заполняется автоматически, если теги копируются в ручную то требуется задатать свойство Text - имя тега для тренда
   "2080TN450A01Z01.DQ.AL_H3" : Bool AT %DB5128.DBX16.0, 500 ms
   "2080TN450A01Z01.DQ.AL_H2" : Bool AT %DB5128.DBX16.1, 500 ms
   "2080TN450A01Z01.DQ.AL_H1" : Bool AT %DB5128.DBX16.2, 500 ms
   "2080TN450A01Z01.DQ.AL_L1" : Bool AT %DB5128.DBX16.3, 500 ms
   "2080TN450A01Z01.DQ.AL_L2" : Bool AT %DB5128.DBX16.4, 500 ms
   "2080TN450A01Z01.DQ.AL_L3" : Bool AT %DB5128.DBX16.5, 500 ms
   "2080TN450A01Z01.DQ.SIG_OK" : Bool AT %DB5128.DBX16.6, 500 ms
   "2080TN450A01Z01.DQ.LIM_H2" : Bool AT %DB5128.DBX16.7, 500 ms
   "2080TN450A01Z01.DQ.LIM_H1" : Bool AT %DB5128.DBX17.0, 500 ms
   "2080TN450A01Z01.DQ.LIM_L1" : Bool AT %DB5128.DBX17.1, 500 ms
   "2080TN450A01Z01.DQ.LIM_L2" : Bool AT %DB5128.DBX17.2, 500 ms
   "2080TN450A01Z01.DQ.GR_P" : Bool AT %DB5128.DBX17.3, 500 ms
   "2080TN450A01Z01.DQ.GR_N" : Bool AT %DB5128.DBX17.4, 500 ms
   "2080TN450A01Z01.I.IN" : Real AT %DB5128.DBD2, 500 ms
   "2080TN450A01Z01.I.SIG_TYPE" : Int AT %DB5128.DBW0, 500 ms
   "2080TN450A01Z01.I.FI_BUS" : Byte AT %DB5128.DBB6, 500 ms
   "2080TN450A01Z01.DI.U_RANGE" : Bool AT %DB5128.DBX7.0, 500 ms
   "2080TN450A01Z01.DI.O_RANGE" : Bool AT %DB5128.DBX7.1, 500 ms
   "2080TN450A01Z01.DI.SIG_FAULT" : Bool AT %DB5128.DBX7.2, 500 ms
   "2080TN450A01Z01.DI.EnConfig" : Bool AT %DB5128.DBX7.3, 500 ms
   "2080TN450A01Z01.DI.AEN" : Bool AT %DB5128.DBX7.4, 500 ms
   "2080TN450A01Z01.DI.AL_SUPR" : Bool AT %DB5128.DBX7.5, 500 ms
   "2080TN450A01Z01.Q.PV_NORM" : Real AT %DB5128.DBD8, 500 ms
   "2080TN450A01Z01.Q.PV_SCAL" : Real AT %DB5128.DBD12, 500 ms
   "2080TN450A01Z01.ParentInfo" : TextRef, internal   // Имя родителя для попап окна, вкладка инфо. При експорте из ECS через скрипт заполняется автоматически, если теги копируются в ручную то требуется в ручную задатать свойство Start Value

